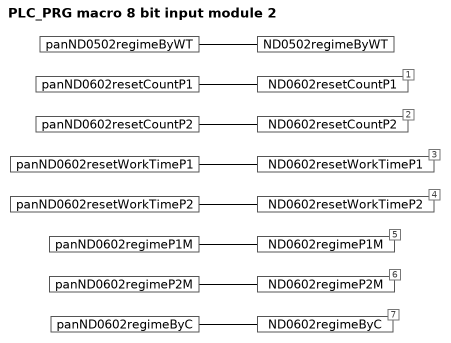
[picture p72: PLC_PRG macro 8 bit input module 2 (CFC)]
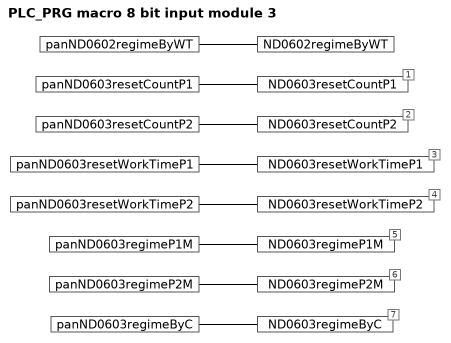
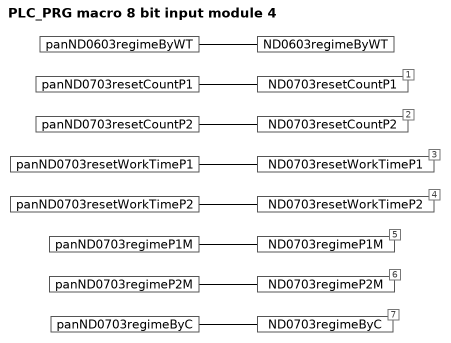
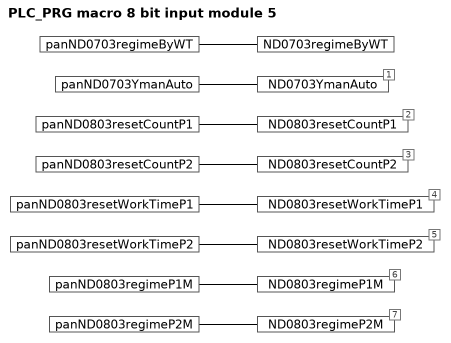
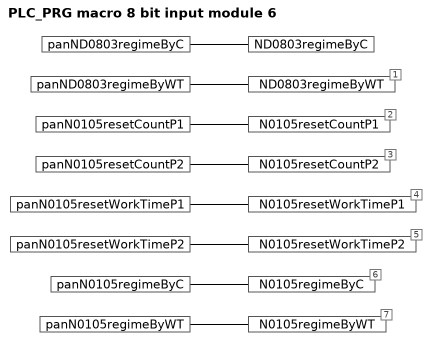
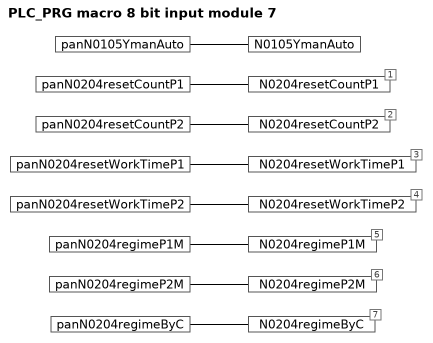
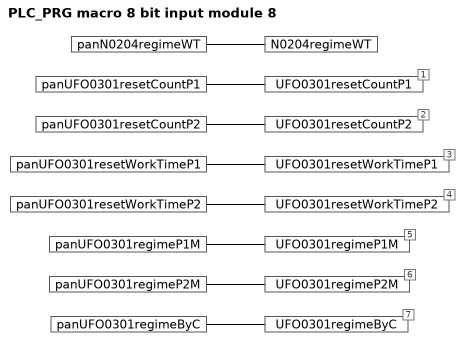
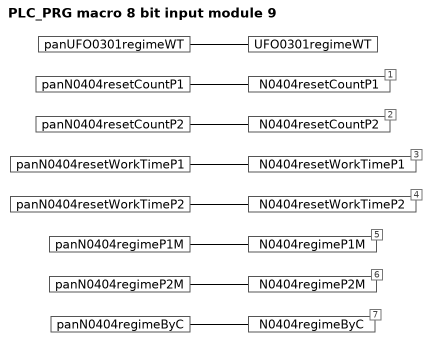
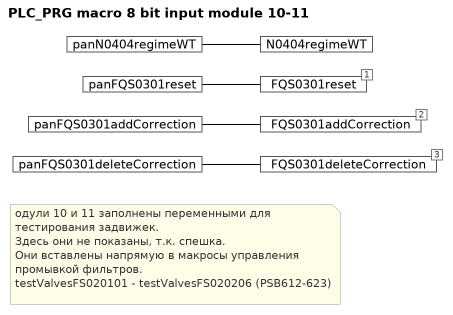
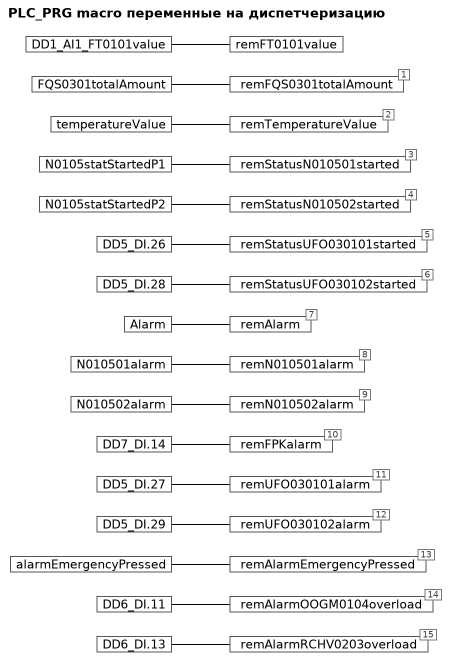
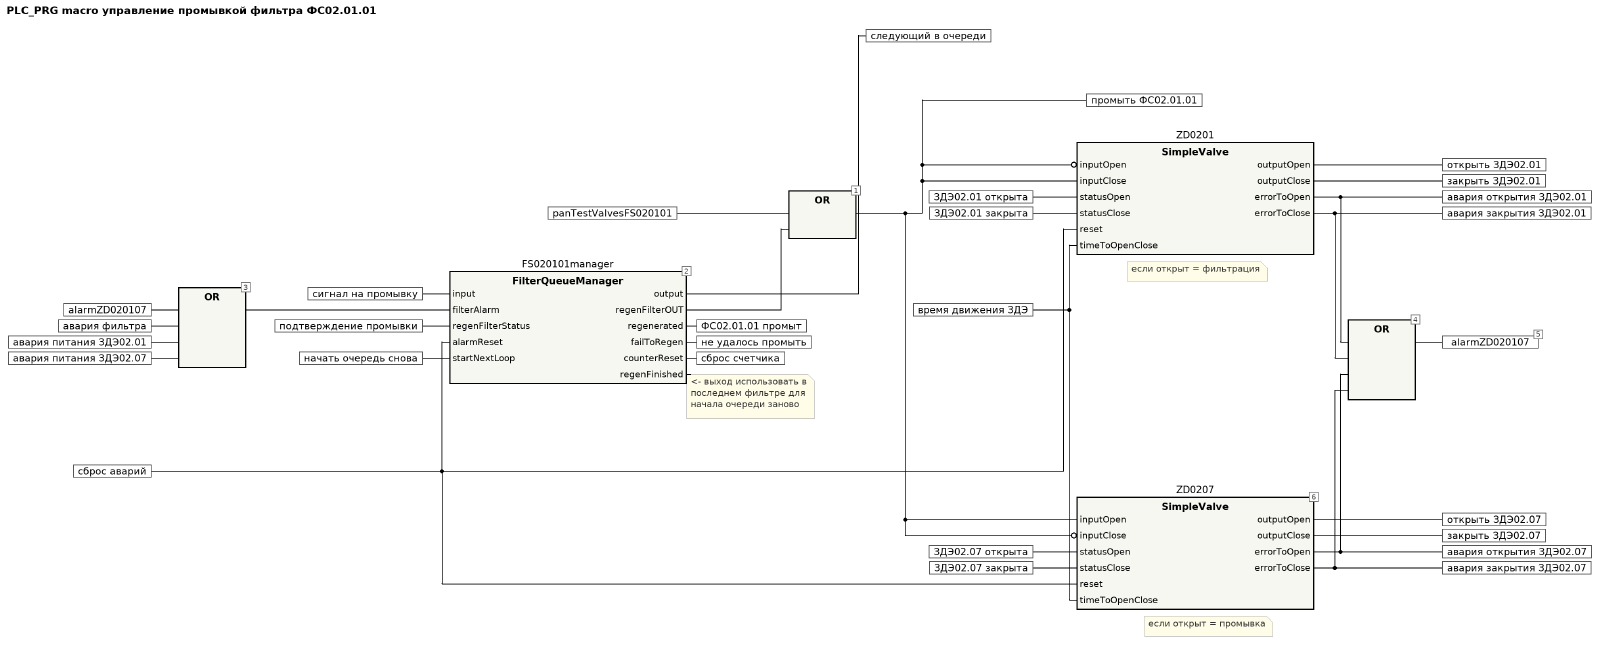
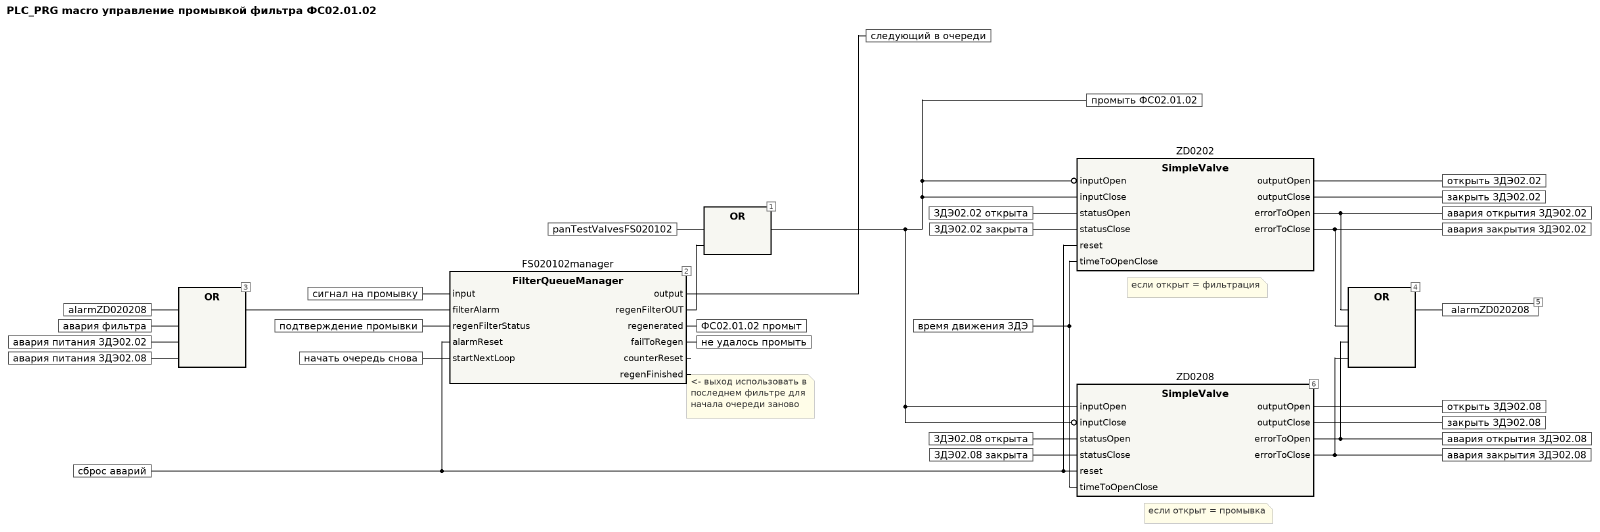
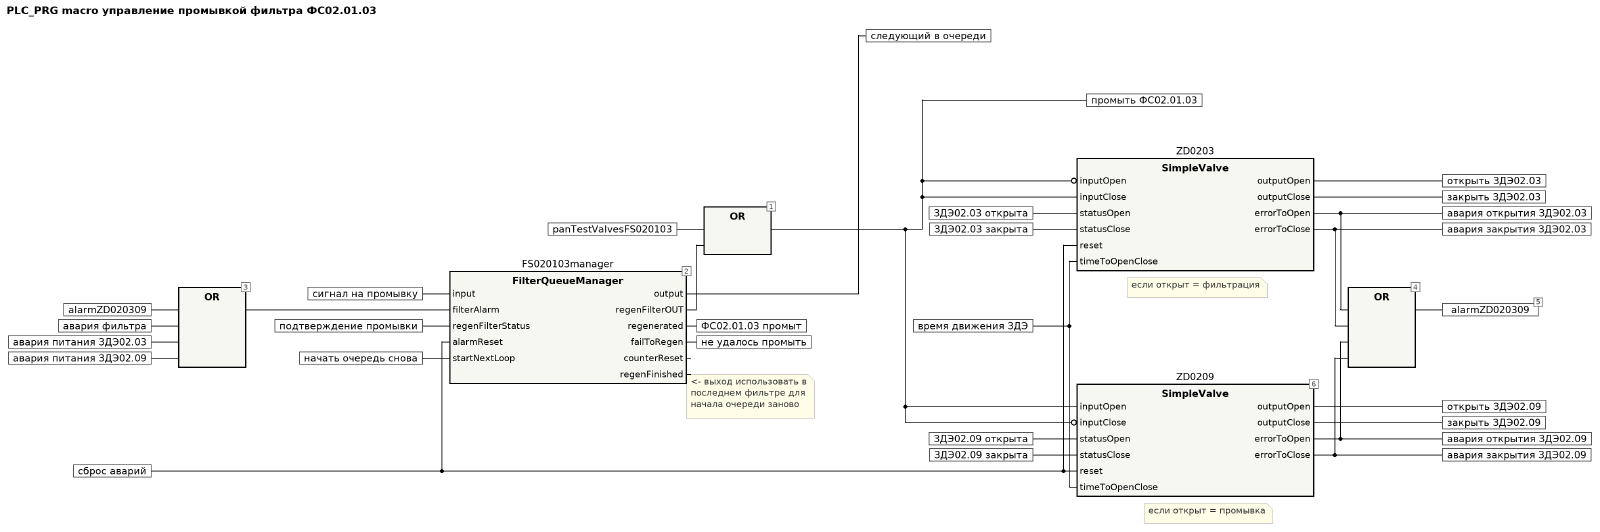
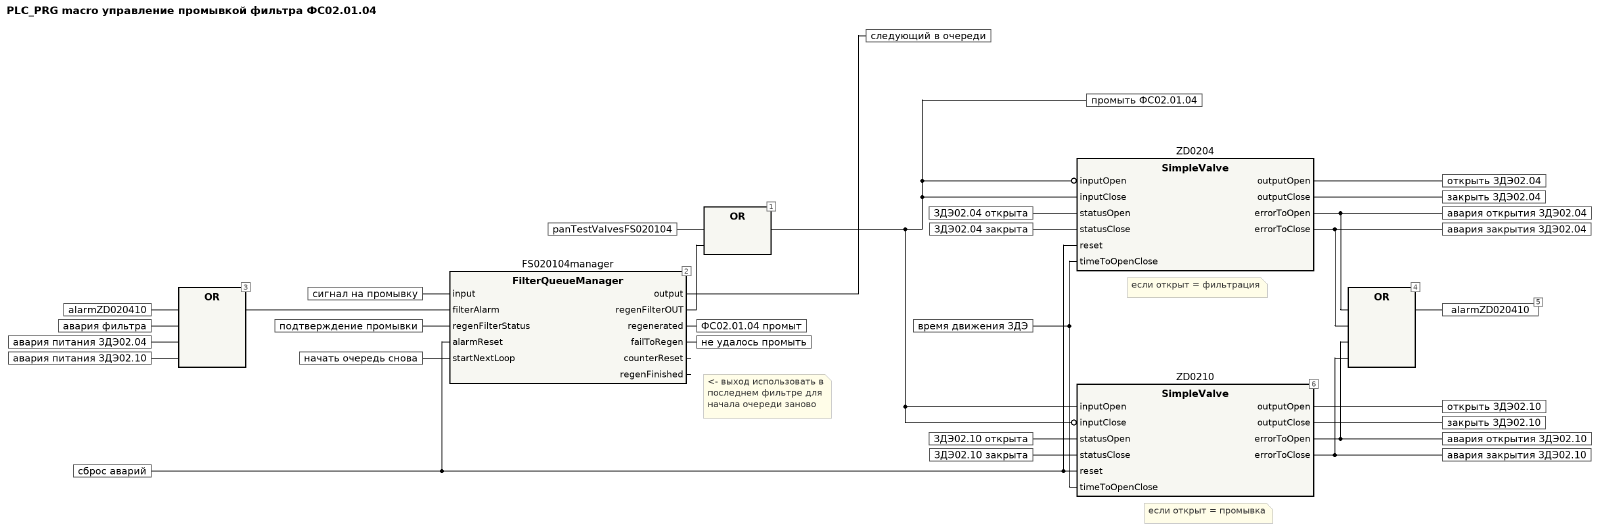
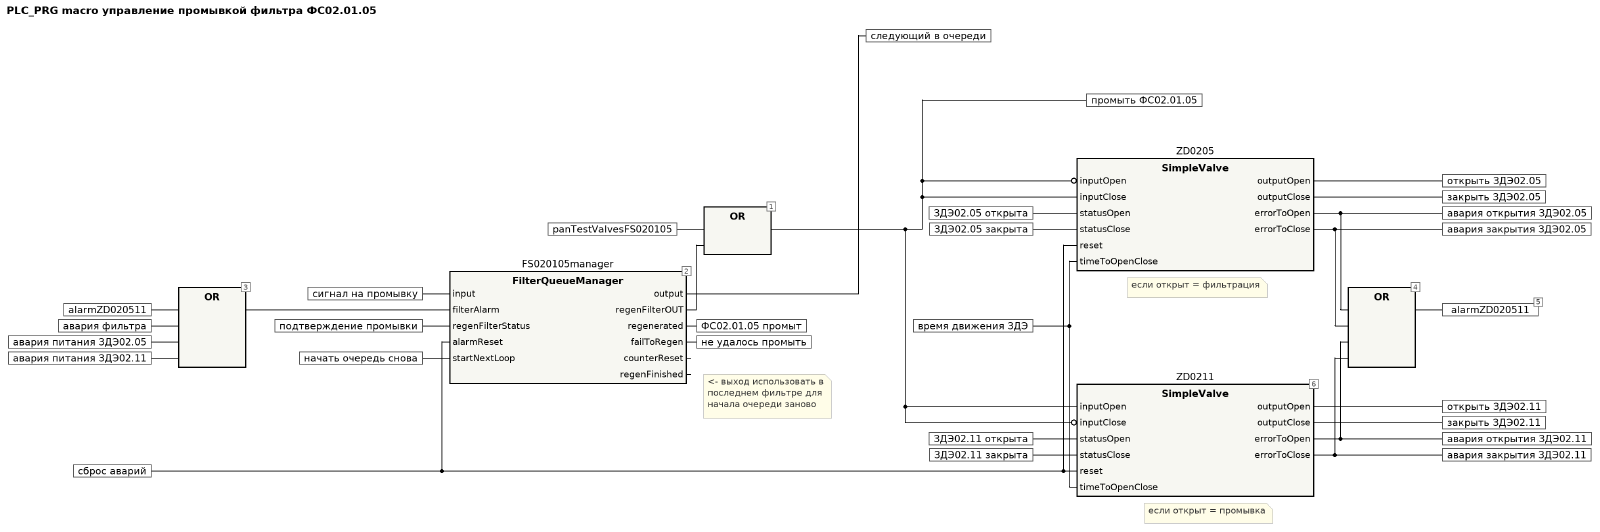
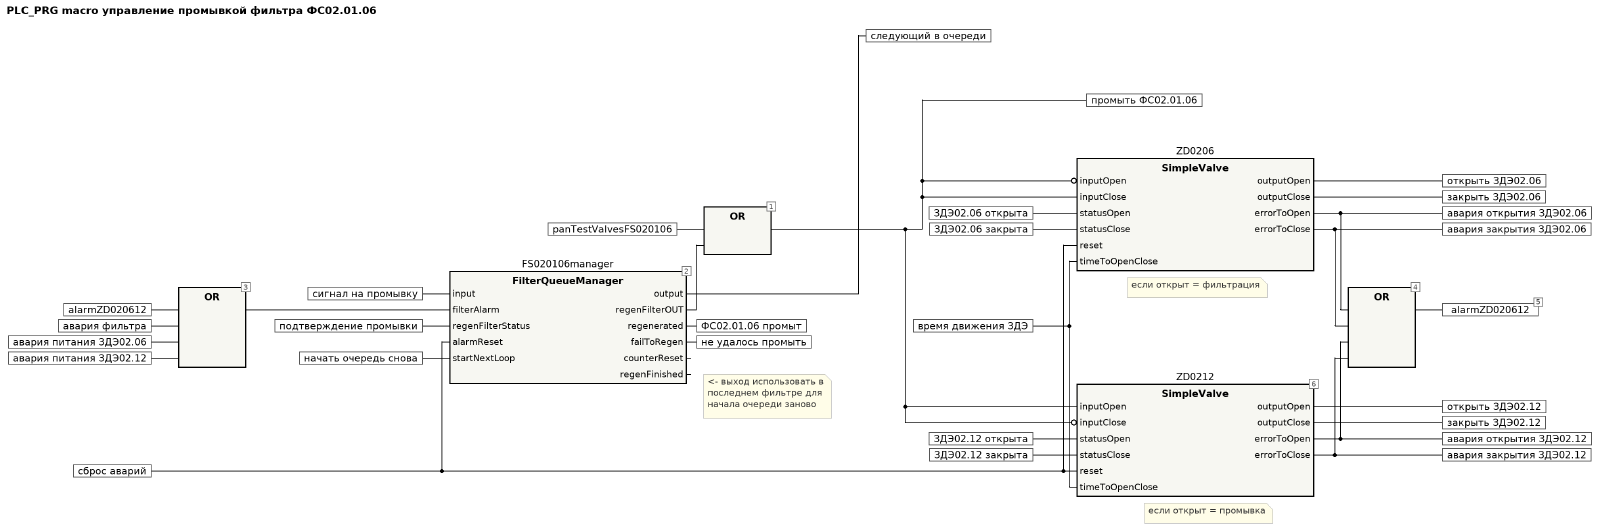
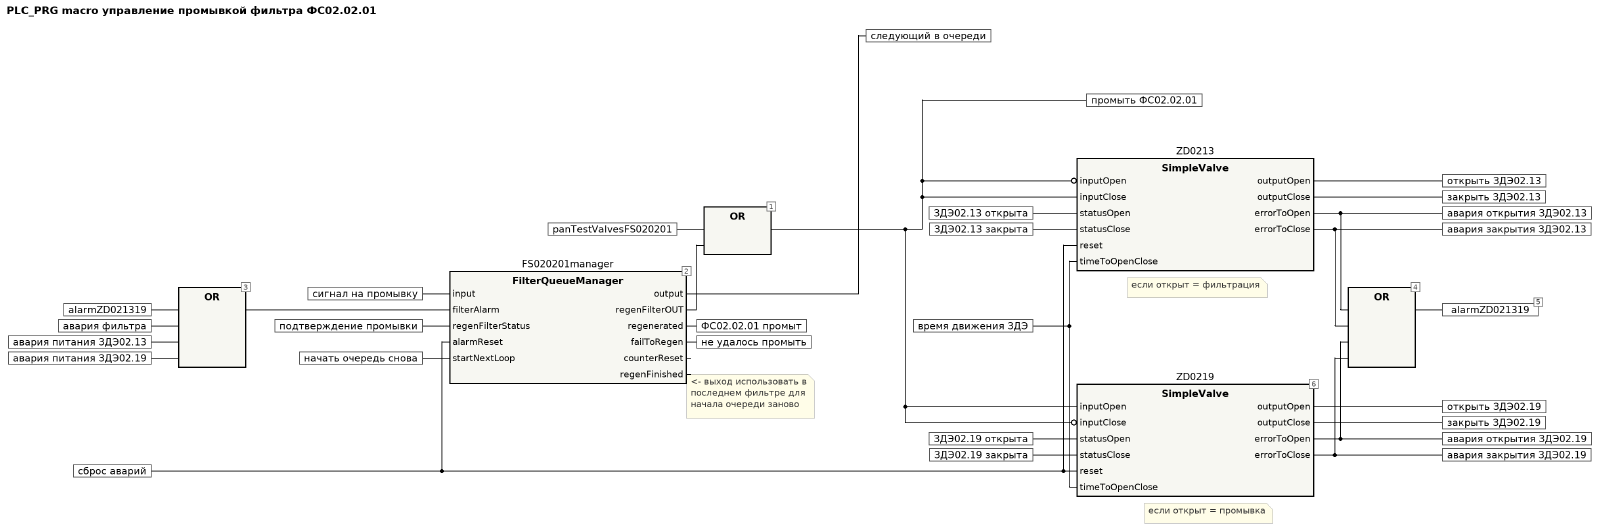
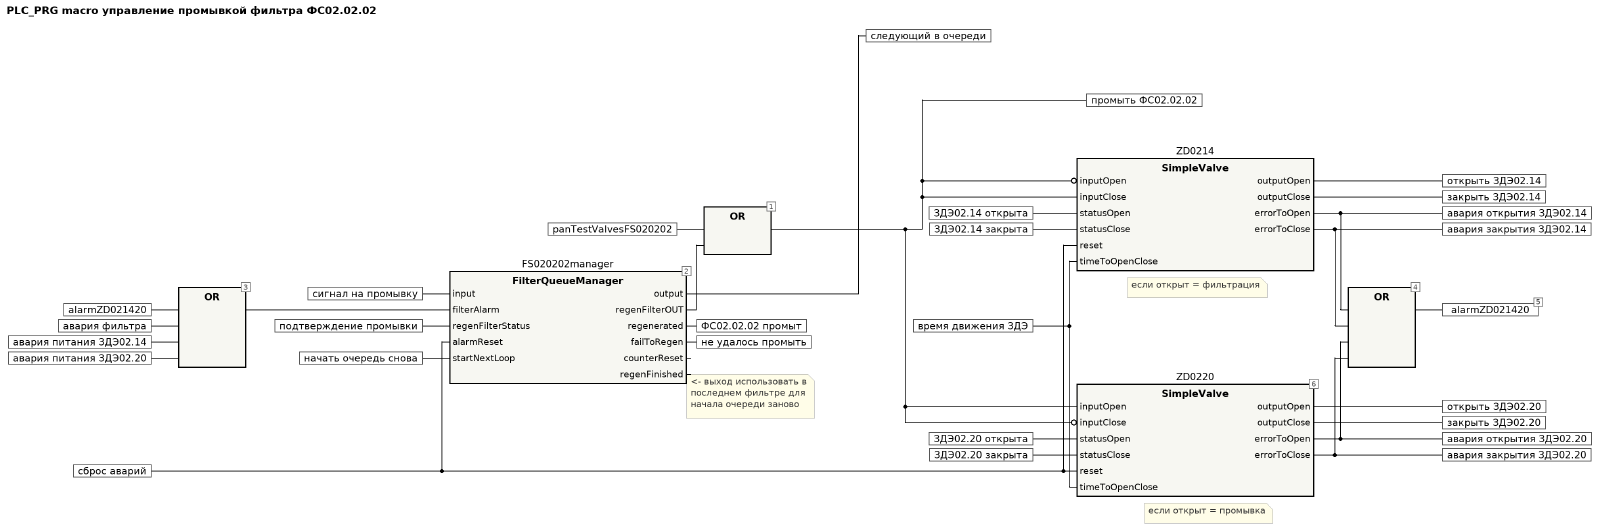
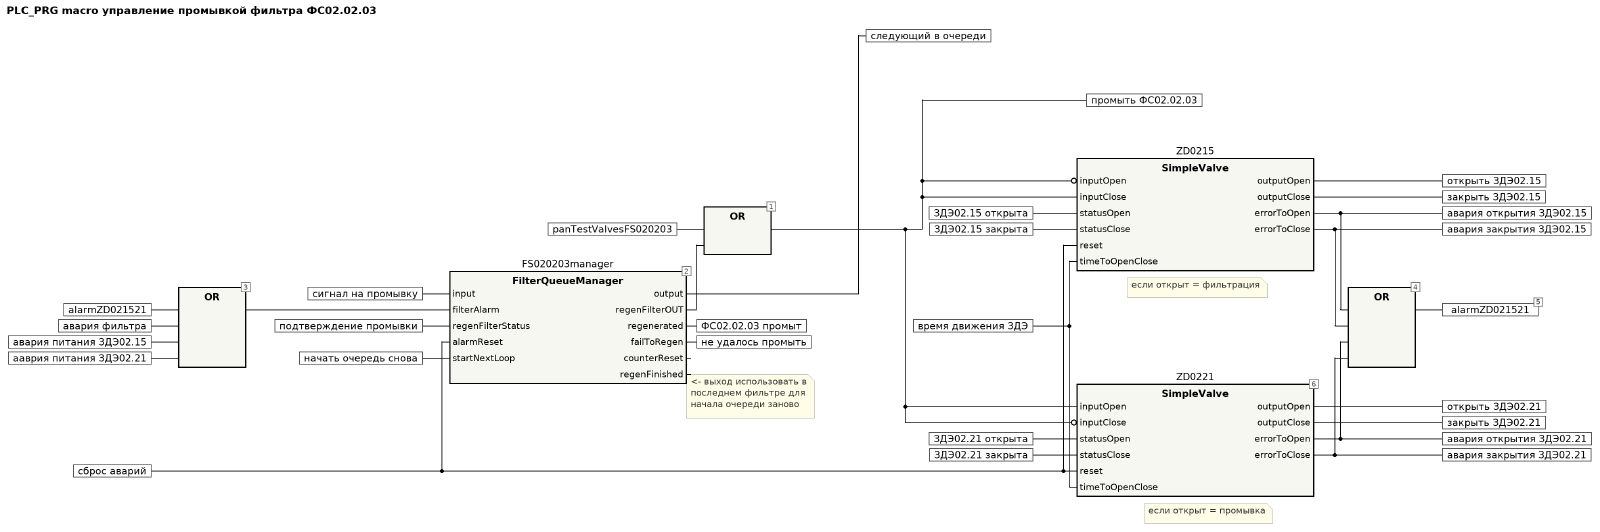
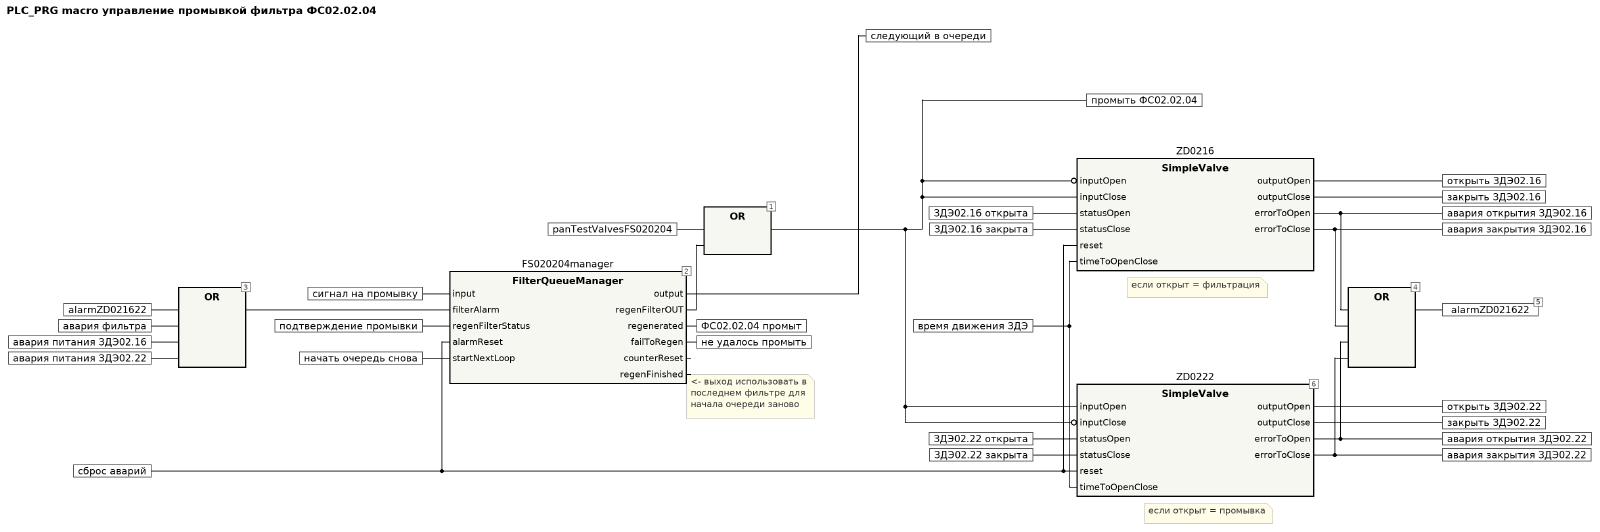
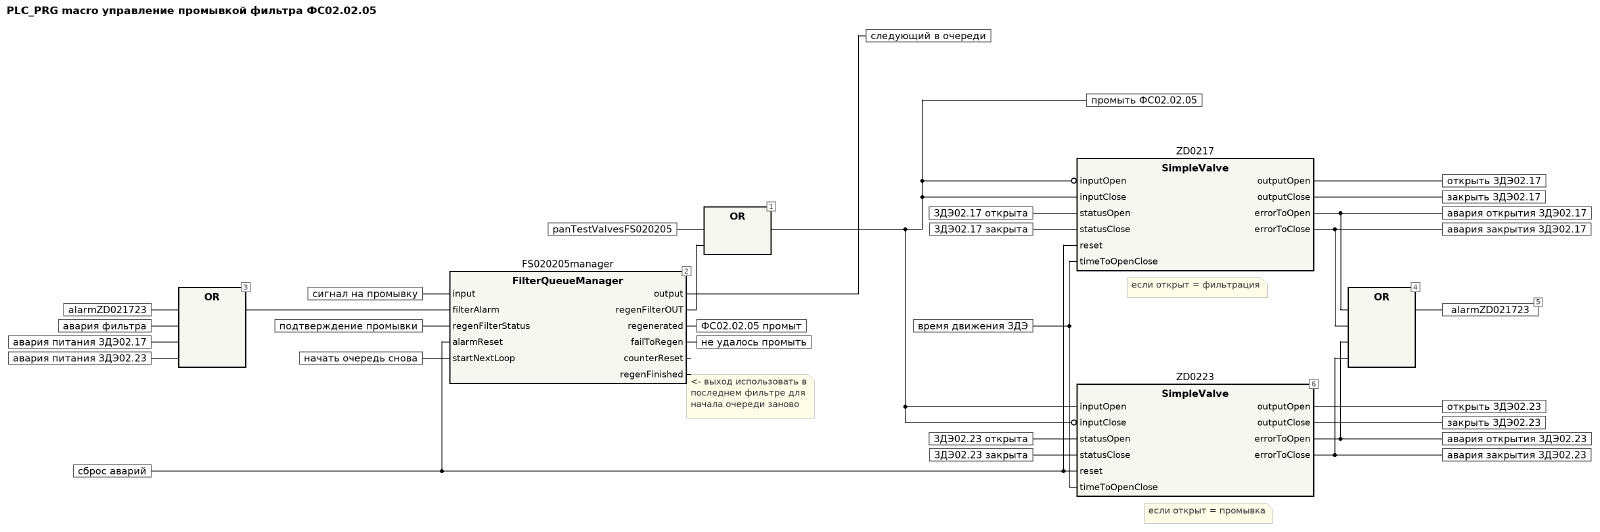
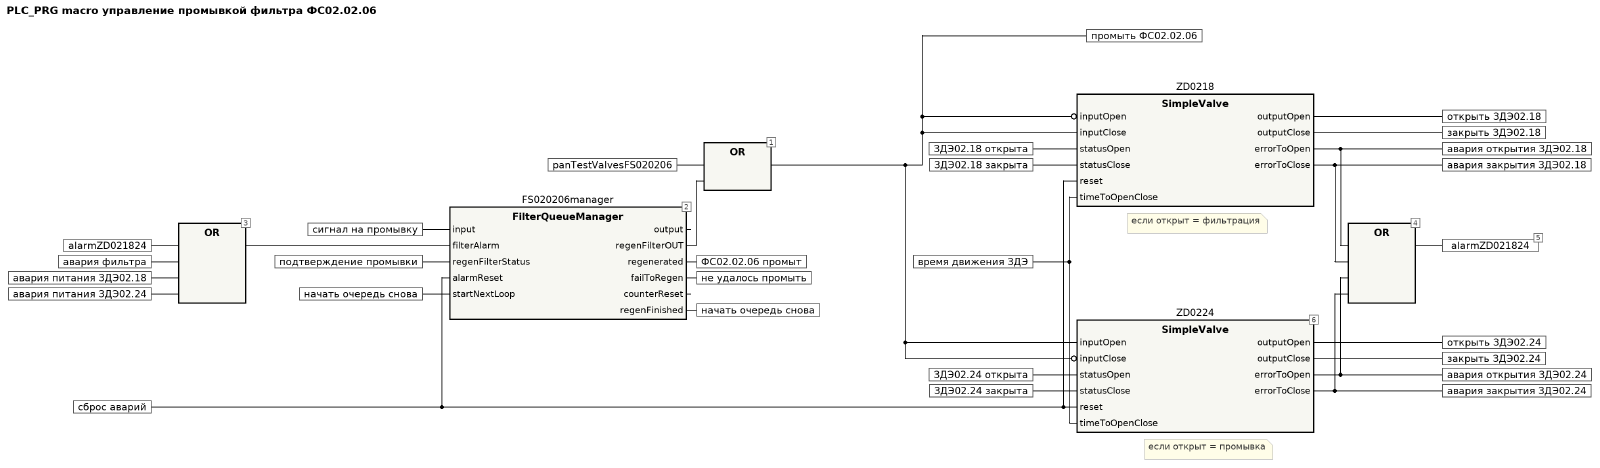
_CFC_ (* Continuous Function Chart, elements in execution order *)
(* 0 = перелив *)
(* авария обоих УФО, если проблемы / открытия/закрытия на одной из задвижек *)
(* авария питания ЗДЭ03.02 *)
(* авария питания ЗДЭ03.01 *)
(* статус-пуск Н01.05/02 *)
(* вкл КМ3 *)
(* Статус ПУСК / ЧРП Н01.05 *)
(* статус-пуск Н01.05/01 *)
(* вкл КМ2 *)
(* контроль обрыва или ошибок модулей в сети ПЛК *)
(* LSA01.02 перелив ОГМ01.04 *)
(* Нажат аварийный стоп. *)
(* авария сети (РКФ) *)
(* разрешение работы КНС / 1 = разрешено *)
(* Нажат аварийный стоп. *)
(* Блок управления разрешением работы КНС *)
(* авария сети (РКФ) *)
(* Авария питания клапанов КЭМ. *)
(* Авария питания розеток / управл.клапанов фильтров. *)
(* авария КНС *)
(* блок подачи сигнала на промывку *)
(* суммируем каждую секунду значение / мгновенного расхода в кубометрах в секунду *)
(* преобразуем расход из / кубометров в час в / кубометры в секунду *)
(* если есть расход / (больше нуля) *)
(* выдает импульс / каждую секунду *)
(* здесь мгновенный расход / в кубометрах в час (FT01.02) *)
(* Авария Н02.04/01 (0=авария) *)
(* Авария Н02.04/02 (0=авария) *)
(* промывка ФС02.01/06 *)
(* промывка ФС02.01/05 *)
(* промывка ФС02.01/04 *)
(* промывка ФС02.01/03 *)
(* промывка ФС02.01/02 *)
(* промывка ФС02.01/01 *)
(* пуск/стоп НД08.03/01 *)
(* пуск/стоп НД08.03/02 *)
(* пуск/стоп НД06.03/01 *)
(* пуск/стоп НД06.03/02 *)
(* пуск/стоп НД06.02/01 *)
(* пуск/стоп НД06.02/02 *)
(* пуск/стоп НД08.04 *)
(* пуск/стоп НД07.03/01 *)
(* пуск/стоп НД07.03/02 *)
(* авария М08.02 (УПФ) *)
(* авария М07.02 (УПЩ) *)
(* авария М06.04 (УПК) *)
(* работа М08.02 (УПФ) *)
(* работа М07.02 (УПЩ) *)
(* работа М06.04 (УПК) *)
(* Контроль, если УФО включили вручную, / а потока при этом нет. *)
(* авария УФО03.01/02 *)
(* работа УФО03.01/02 *)
(* авария УФО03.01/01 *)
(* Для подачи предостережения на пульте / оператора (при необходимости), а также / сигнализации лампой АВАРИЯ. *)
(* работа УФО03.01/01 *)
(* авария УФО03.01/02 *)
(* авария УФО03.01/01 *)
(* авария Н04.04/01 *)
(* авария Н04.04/02 *)
(* время контроля старта ФПК (по умолч.=3мин) *)
(* время работы ФПК после спада сигнала датч.осадка *)
(* запуск фильтрации *)
(* Защита от сухого хода насоса ФПК *)
(* датчик уровня осадка *)
(* Давление на входе ФПК (0...16 бар) *)
(* авария ФПК *)
(* подающий насос ФПК работает *)
(* ФПК готов к приему *)
(* ФПК не запустился *)
(* рН-метр QE01.02 на входе, / диапазон 0...14 *)
(* авария входа рН-метра QE01.01 *)
(* авария входа расходомера FT01.02 *)
(* расходомер FT01.01 на входе, / диапазон 0...600куб/час *)
(* авария НД08.04 *)
(* управление 4...20мА НД08.03/01 *)
(* пуск/стоп НД08.03/01 *)
(* пуск/стоп НД08.03/02 *)
(* управление 4...20мА НД08.03/02 *)
(* авария привода НД08.03/01 *)
(* авария привода НД08.03/02 *)
(* авария НД07.03/01 *)
(* авария НД07.03/02 *)
(* управление 4...20мА НД07.03/01 *)
(* управление 4...20мА НД07.03/02 *)
(* пуск/стоп НД07.03/01 *)
(* пуск/стоп НД07.03/02 *)
(* авария НД07.03/01 *)
(* авария НД07.03/02 *)
(* авария НД06.03/01 *)
(* авария НД06.03/02 *)
(* авария НД06.02/01 *)
(* авария НД06.02/02 *)
(* управление 4...20мА НД06.03/01 *)
(* пуск/стоп НД06.03/01 *)
(* пуск/стоп НД06.03/02 *)
(* управление 4...20мА НД06.03/02 *)
(* авария НД06.03/01 *)
(* авария НД06.03/02 *)
(* управление 4...20мА НД06.02/01 *)
(* пуск/стоп НД06.02/01 *)
(* пуск/стоп НД06.02/02 *)
(* управление 4...20мА НД06.02/02 *)
(* авария НД06.02/01 *)
(* авария НД06.02/02 *)
(* ошибка блока дозирования НД05.02 *)
(* авария входа датчика температуры *)
(* лампа АВАРИЯ *)
(* датчик температуры в помещении / (метран) диапазон: 0...+100С *)
(* управление 4...20мА НД05.02/01 *)
(* пуск/стоп НД05.02/01 *)
(* авария НД05.02/01 *)
(* авария НД05.02/02 *)
(* пуск/стоп НД05.02/02 *)
(* управление 4...20мА НД05.02/02 *)
(* АВАРИИ *)
(* авария привода НД08.03/01 *)
(* авария привода НД08.03/02 *)
(* авария НД08.04 *)
(* насос Н04.01 работает *)
(* пуск/стоп НД08.04 *)
(* управление 4...20мА НД08.04 *)
(* авария входа расходомера FT01.01 *)
(* расходомер FT01.02 на входе, / диапазон 0...600куб/час *)
(* рН-метр QE01.01 на входе, / диапазон 0...14 *)
(* авария входа рН-метра QE01.02 *)
(* сухой ход НД08.03/01 *)
(* сухой ход НД08.03/02 *)
(* сухой ход НД08.03/01 *)
(* сухой ход НД08.03/02 *)
(* LSA01.02 перелив ОГМ01.04 *)
(* Инициализирует требуемые булевые переменные / в момент старта выполнения программы. *)
(* Статус ПУСК ЧРП Н01.05 *)
(* LS01.03 - рабочий верхний уровень ОГМ01.04 автоматический пуск 01.05 *)
(* LS01.04 - нижний уровень ОГМ01.04, сухой ход Н01.05 *)
(* SA1 Ручной выбор Н01.05/01 = главный *)
(* SA1 Ручной выбор Н01.05/02 = главный *)
(* Стоп  Н01.05 (сброс самоподхвата реле) *)
(* время на создание потока *)
(* Пуск  Н01.05 *)
(* КМ1 питание ЧРП *)
(* КМ2 питание насоса 1 *)
(* КМ3 питание насоса 2 *)
(* Авария ЧРП Н01.05 *)
(* термоконтакт Н01.05/01 *)
(* термоконтакт Н01.05/02 *)
(* авария питания ЗДЭ02.25 *)
(* LSА02.01 Перелив РЧВ02.03 *)
(* Давление на входе ФПК / 0...16 бар (мах допуст.10) *)
(* Авария входа AI6 ПЛК, давл.ФПК *)
(* авария ФПК *)
(* Открыть КШЭ04.01 *)
(* статус КШЭ04.01 открыт *)
(* Закрыть КШЭ04.01 *)
(* статус КШЭ04.01 закрыт *)
(* подающий насос ФПК работает *)
(* стоп Н04.04 *)
(* пуск Н04.04/02 *)
(* пуск Н04.04/01 *)
(* авт.пуск Н04.04 *)
(* сухой ход Н04.04, 0=защита *)
(* авария Н04.04/01, 0=авария *)
(* авария Н04.04/02, 0=авария *)
(* импульсный расходомер *)
(* Авария Н02.04/01 (0=авария) *)
(* Авария Н02.04/02 (0=авария) *)
(* промывка ФС02.02/06 *)
(* промывка ФС02.02/05 *)
(* промывка ФС02.02/04 *)
(* промывка ФС02.02/03 *)
(* промывка ФС02.02/02 *)
(* промывка ФС02.02/01 *)
(* Клапан КЭМ05.01 открыт. *)
(* Клапан КЭМ06.01 открыт. *)
(* Клапан КЭМ07.01 открыт. *)
(* Клапан КЭМ08.01 открыт. *)
(* Сухой ход Н02.04 (LS02.03) 0=сух.ход *)
(* Стоп Н02.04, / сброс самоподхвата реле, / пока активно пуск - невозможен *)
(* Пуск Н02.04/01 *)
(* Пуск Н02.04/02 *)
(* текущий объем *)
(* заданный до промывки объем *)
(* 0=авария *)
(* авария (при 0) ФС02.01/06 *)
(* авария (при 0) ФС02.01/05 *)
(* авария (при 0) ФС02.01/04 *)
(* авария (при 0) ФС02.01/03 *)
(* авария (при 0) ФС02.01/02 *)
(* авария (при 0) ФС02.01/01 *)
(* авария (при 0) ФС02.02/06 *)
(* авария (при 0) ФС02.02/05 *)
(* авария (при 0) ФС02.02/04 *)
(* авария (при 0) ФС02.02/03 *)
(* авария (при 0) ФС02.02/02 *)
(* авария (при 0) ФС02.02/01 *)
(* сброс счетчика стоков до следующей промывки *)
(* подсчет общего объема стоков, прошедшего через расходомер FT01.02 *)
(* очередь передается на 2 ступень *)
(* авария питания ЗДЭ02.01 *)
(* авария питания ЗДЭ02.02 *)
(* авария питания ЗДЭ02.03 *)
(* авария питания ЗДЭ02.04 *)
(* авария питания ЗДЭ02.05 *)
(* авария питания ЗДЭ02.06 *)
(* авария питания ЗДЭ02.07 *)
(* авария питания ЗДЭ02.08 *)
(* авария питания ЗДЭ02.09 *)
(* авария питания ЗДЭ02.10 *)
(* авария питания ЗДЭ02.11 *)
(* авария питания ЗДЭ02.12 *)
(* авария питания ЗДЭ02.13 *)
(* авария питания ЗДЭ02.14 *)
(* авария питания ЗДЭ02.15 *)
(* авария питания ЗДЭ02.16 *)
(* авария питания ЗДЭ02.17 *)
(* авария питания ЗДЭ02.18 *)
(* авария питания ЗДЭ02.19 *)
(* авария питания ЗДЭ02.20 *)
(* авария питания ЗДЭ02.21 *)
(* авария питания ЗДЭ02.22 *)
(* авария питания ЗДЭ02.23 *)
(* авария питания ЗДЭ02.24 *)
(* инвертирование сигнала, чтобы все аварии / обозначались как 1 (TRUE) *)
(* авария НД05.02/01 *)
(* авария НД05.02/02 *)
(* авария питания КШЭ04.01 *)
(* 1=открыть; 0 = закрыть *)
(* в этом макросе лежит управление режимом тестирования задвижек ЗДЭ03 / Тестирование запрещает автоматический запуск УФО от ПЛК *)
(* стоп от / панели оператора *)
#0 rTrigStartInitializer:R_TRIG(CLK: TRUE)
#1 startInitializer <= #0.Q
#2 MACRO контроль температуры в помещении(pin 1 "вход датчика температуры": DD1_AI0, pin 2 "минимально допустимая температура в помещении": maxTemperature, pin 3 "максимально допустимая температура в помещении": minTemperature)
	(* задаем границы допустимой температуры в помещении / проверяем что измеренное значение в заданном диапазоне *)
	(* не смотрим конкретный тип ошибки / (работает не точно, обрыв определяет как слишком маленькое значение) / если не равно 0 - значит на входе ошибка *)
	#3 DD1_AI0_temperature:DECODE_FLOAT(VALUE: pin 1, DEF_VALUE: -)
	#4 NE(#3._ERR, 0)
	out 2 "авария датчика температуры" <= #4
	out 1 "температура в помещении" <= #3.OUT_VALUE
	#5 REAL_TO_INT(#3.OUT_VALUE)
	#6 temperatureLimits:LIMITALARM(IN: #5, HIGH: pin 3, LOW: pin 2)
	out 3 "температура выше заданного диапазона" <= #6.O
	out 4 "температура ниже заданного диапазона" <= #6.U
	#7 temperatureLimits:LIMITALARM(IN: -, HIGH: -, LOW: -)
END_MACRO
#8 temperatureValue <= #2.out 1
#9 DD1_AI0_error <= #2.out 2
#10 alarmHighTemperature <= #2.out 3
#11 alarmLowTemperature <= #2.out 4
#12 OR(testKSHE0401, DD7_DI.13)
#13 MACRO клапан шаровый перед ФПК (КШЭ04.01)(pin 1 "сигнал "подающий насос ФПК" работает": #12, pin 2 "статус КШЭ04.01 открыт": DD9_DI.2, pin 3 "статус КШЭ04.01 закрыт": DD9_DI.3, pin 4 "сброс аварий": alarmReset, pin 5 "время на открытие/закрытие": timeToOpenCloseValve)
	#14 FPKkshe0401DelayToOpen:TON(IN: #16.outputOpen, PT: T#1s)
	out 1 "выход на открытие КШЭ04.01" <= #14.Q
	#15 FPKkshe0401DelayToClose:TON(IN: #16.outputClose, PT: T#1s)
	out 2 "выход на закрытие КШЭ04.01" <= #15.Q
	#16 FPKkshe0401:SimpleValve(inputOpen: pin 1, inputClose: #17, statusOpen: pin 2, statusClose: pin 3, reset: pin 4, timeToOpenClose: pin 5)
	#17 NOT(pin 1)
	out 3 "авария на открытие КШЭ04.01" <= #16.errorToOpen
	out 4 "авария на закрытие КШЭ04.01" <= #16.errorToClose
END_MACRO
#18 DD4_DO.2 <= #13.out 1
#19 DD4_DO.3 <= #13.out 2
#20 FPKkshe0401errorToOpen <= #13.out 3
#21 FPKkshe0401errorToClose <= #13.out 4
#22 OR(DD1_AI0_error, DD1_AI1_error, DD1_AI2_error, DD1_AI3_error, DD1_AI4_error, alarmHighTemperature, alarmLowTemperature, ND0502dosingError, ND0602dosingError, ND0603dosingError, ND0803dosingError, ND0804dosingError, DD1_DI6, DD1_DI7, N010501alarm, N010502alarm, ZDE0225errorToOpen, ZDE0225errorToClose, DD7_DI.14, FPKnotStarted, DD1_AI5_error, FPKkshe0401errorToOpen, FPKkshe0401errorToClose, DD5_DI.27, DD5_DI.29, filterFailToRegen020101, errorToOpenZD0201, errorToCloseZD0201, errorToOpenZD0207, errorToCloseZD0207, filterFailToRegen020102, errorToOpenZD0202, errorToCloseZD0202, errorToOpenZD0208, errorToCloseZD0208, filterFailToRegen020103, errorToOpenZD0203, errorToCloseZD0203, errorToOpenZD0209, errorToCloseZD0209, filterFailToRegen020104, errorToOpenZD0204, errorToCloseZD0204, errorToOpenZD0210, errorToCloseZD0210, filterFailToRegen020105, errorToOpenZD0205, errorToCloseZD0205, errorToOpenZD0211, errorToCloseZD0211, filterFailToRegen020106, errorToOpenZD0206, errorToCloseZD0206, errorToOpenZD0212, errorToCloseZD0212, filterFailToRegen020201, errorToOpenZD0213, errorToCloseZD0213, errorToOpenZD0219, errorToCloseZD0219, filterFailToRegen020202, errorToOpenZD0214, errorToCloseZD0214, errorToOpenZD0220, errorToCloseZD0220, filterFailToRegen020203, errorToOpenZD0215, errorToCloseZD0215, errorToOpenZD0221, errorToCloseZD0221, filterFailToRegen020204, errorToOpenZD0216, errorToCloseZD0216, errorToOpenZD0222, errorToCloseZD0222, filterFailToRegen020205, errorToOpenZD0217, errorToCloseZD0217, errorToOpenZD0223, errorToCloseZD0223, filterFailToRegen020206, errorToOpenZD0218, errorToCloseZD0218, errorToOpenZD0224, errorToCloseZD0224, alarmPLKnetwork, alarmND050201, alarmND050202, alarmND060201, alarmND060202, alarmND060301, alarmND060302, alarmND070301, alarmND070302, alarmND080301, alarmND080302, alarmND0804, alarmOGM0104overload, alarmRCHV0203overload, alarmN040402, alarmN040401, alarmM0604, alarmM0702, alarmM0802, alarmN020401, alarmN020402, alarmFS020101, alarmFS020102, alarmFS020103, alarmFS020104, alarmFS020105, alarmFS020106, alarmFS020201, alarmFS020202, alarmFS020203, alarmFS020204, alarmFS020205, alarmFS020206, alarmZDE0201power, alarmZDE0202power, alarmZDE0203power, alarmZDE0204power, alarmZDE0205power, alarmZDE0206power, alarmZDE0207power, alarmZDE0208power, alarmZDE0209power, alarmZDE0210power, alarmZDE0211power, alarmZDE0212power, alarmZDE0213power, alarmZDE0214power, alarmZDE0215power, alarmZDE0216power, alarmZDE0217power, alarmZDE0218power, alarmZDE0219power, alarmZDE0220power, alarmZDE0221power, alarmZDE0222power, alarmZDE0223power, alarmZDE0224power, alarmZDE0225power, alarmKSHE0401power, alarmKNS, alarmPowerSocketFS, alarmKEMvalvesPower, alarmEmergencyPressed, alarmRKF, errorToOpenZDE0301, errorToCloseZDE0301, errorToOpenZDE0302, errorToCloseZDE0302, alarmZDE0301power, alarmZDE0302power)
#23 DD1_DO11 <= #22
#24 alarm <= #22
#25 MACRO контроль аналогового входа DD1_AI1(pin 1 "вход": DD1_AI1)
	(* Не смотрим конкретную ошибку, / определяем,что вход неисправен без расшифровки. *)
	#26 DD1_AI1_FT0101:DECODE_FLOAT(VALUE: pin 1, DEF_VALUE: -)
	#27 NE(#26._ERR, 0)
	out 2 "авария" <= #27
	out 1 "выход" <= #26.OUT_VALUE
END_MACRO
#28 DD1_AI1_FT0101value <= #25.out 1
#29 DD1_AI1_error <= #25.out 2
#30 MACRO контроль аналогового входа DD1_AI2(pin 1 "вход": DD1_AI2)
	(* Не смотрим конкретную ошибку, / определяем,что вход неисправен без расшифровки. *)
	#31 DD1_AI2_FT0102:DECODE_FLOAT(VALUE: pin 1, DEF_VALUE: -)
	#32 NE(#31._ERR, 0)
	out 2 "авария" <= #32
	out 1 "выход" <= #31.OUT_VALUE
END_MACRO
#33 DD1_AI2_FT0102value <= #30.out 1
#34 DD1_AI2_error <= #30.out 2
#35 MACRO управление Н01.05 (поддержание заданного расхода по FT01.02)(pin 1 "статус ПУСК ЧРП (реле)": DD5_DI.4, pin 2 "LS01.03 раб.уров.": DD6_DI.12, pin 3 "LS01.04 ниж.уров.(сух.ход)": DD5_DI.0, pin 4 "SA1ручной выб.Н01.05/01-главный": DD5_DI.5, pin 5 "SA1ручной выб.Н01.05/02-главный": DD5_DI.6, pin 6 "включить режим "по кол.вкл."": N0105regimeByC, pin 7 "включить режим "по наработке"": N0105regimeByWT, pin 8 "значение расхода от FT01.02": DD1_AI2_FT0102value, pin 9 "уставка расхода": N0105flowSetValue, pin 10 "время на создание потока": N0105minFlowTime, pin 11 "Р-коэфф.": N0105koeffP, pin 12 "I-коэфф": N0105koeffI, pin 13 "Д-коэфф": N0105koeffD, pin 14 "управление ЧРП в ручн.реж.(4...20мА)": N0105YoutManual, pin 15 "переключатель управление ЧРП РУЧН/АВТ": N0105YmanAuto, pin 16 "мин.допустимый расход": N0105minFlow, pin 17 "термоконтакт Н01.05/01": DD5_DI.2, pin 18 "термоконтакт Н01.05/02": DD5_DI.3, pin 19 "авария ЧРП Н01.05": DD5_DI.1, pin 20 "сброс аварии": alarmReset, pin 21 "сброс кол-ва вкл.Н01.05/01": N0105resetCountP1, pin 22 "сброс кол-ва вкл.Н01.05/02": N0105resetCountP2, pin 23 "сброс наработки Н01.05/01": N0105resetWorkTimeP1, pin 24 "сброс наработки Н01.05/02": N0105resetWorkTimeP2)
	(* время на создание потока *)
	(* Пуск  Н01.05 *)
	(* режимы по количеству включений,  или по наработке / активны если оба входа SA1 не активны *)
	(* управление Н01.05 - поддержание / заданного расхода по FT01.02 *)
	(* по умолчанию при старте программы *)
	(* если на входе true / то нижнее значение, / иначе то, что посередине *)
	(* Если насос создает давление меньше / указанного, то авария. *)
	#36 OR(pin 2, #37.Q)
	#37 N0105startTrig:R_TRIG(CLK: pin 1)
	#38 N0105stopTrig:F_TRIG(CLK: pin 1)
	#39 N0105startTrigg:RS(SET: #36, RESET1: #41)
	#40 N0105regime:choosePumpRegime(start: #39.Q1, pump1Main: pin 4, pump2Main: pin 5, byCounter: #45, byWorkTime: #54)
	out 2 "статус режим "Н01.05/01 - главный"" <= #40.pump1MainActive
	out 3 "статус режим "Н01.05/02 - главный"" <= #40.pump2MainActive
	out 4 "статус режим "по кол-ву вкл."" <= #40.byCounterActive
	#41 OR(#38.Q, #42)
	out 5 "статус режим "по наработке"." <= #40.byWorkTimeActive
	#42 NOT(pin 3)
	#43 NOT(#39.Q1)
	out 1 "СТОП (сброс самоподхвата реле пуска ЧРП)." <= #43
	#44 AND(#53.pump1active, #63)
	out 15 "авария Н01.05/01" <= #47.Q1
	#45 AND(NOT pin 4, NOT pin 5, #51.Q1)
	#46 OR(#44, #52, NOT pin 17)
	#47 N010501alarmTrig:RS(SET: #46, RESET1: pin 20)
	#48 N010501alarm <= #47.Q1
	#49 OR(pin 6, startInitializer)
	#50 N0105regByCinit:R_TRIG(CLK: #49)
	#51 N0105regByCtrig:RS(SET: #50.Q, RESET1: #55.Q)
	#52 AND(#53.pump1active, NOT pin 19)
	#53 N0105twoPumpOneDriveManager:TwoPumpOneDriveManager(startStopPump1: #40.startPump1, startStopPump2: #40.startPump2, alarmPump1: N010501alarm, alarmPump2: N010502alarm, alarmReset: alarmReset, counterStart: #40.startByCounter, Pump1ResetCounter: pin 21, Pump2ResetCounter: pin 22, ValueToResetCounter: -, workTimeStart: #40.startByWorkTime, workTimePump1Reset: pin 23, workTimePump2Reset: pin 24, timeKM1off: -, timeKM23DelayON: -, timeKM23offDelay: -, timeReadyToStartDelay: -)
	out 6 "кол-во включений Н01.05/01" <= #53.counterPump1
	out 7 "кол-во включений Н01.05/02" <= #53.counterPump2
	out 8 "наработка Н01.05/01" <= #53.currentWorkTimePump1
	#54 AND(NOT pin 4, NOT pin 5, #56.Q1)
	out 9 "наработка Н01.05/02" <= #53.currentWorkTimePump2
	out 10 "КМ1-питание ЧРП" <= #53.DriveKM
	#55 N0105regWTinit:R_TRIG(CLK: pin 7)
	#56 N0105regWTtrig:RS(SET: #55.Q, RESET1: #50.Q)
	out 11 "КМ2-питание Н01.05/01" <= #53.pump1KM
	out 12 "КМ3-питание Н01.05/02" <= #53.pump2KM
	out 13 "пуск ЧРП (Н01.05)" <= #53.driveStart
	out 16 "авария Н01.05/02" <= #59.Q1
	#57 AND(NOT pin 19, #53.pump2active)
	#58 OR(#57, #61, NOT pin 18)
	#59 N010502alarmTrig:RS(SET: #58, RESET1: pin 20)
	#60 N010502alarm <= #59.Q1
	#61 AND(#53.pump2active, #63)
	#62 N0105timerminFlow:TON(IN: #53.driveStart, PT: pin 10)
	#63 AND(#62.Q, #64)
	#64 LE(pin 8, pin 16)
	#65 SEL(#53.driveStart, 0, #66.Y)
	out 14 "управление ЧРП (4...20мА)" <= #65
	#66 N0105pidReg:PID(ACTUAL: pin 8, SET_POINT: pin 9, KP: pin 11, TN: pin 12, TV: pin 13, Y_MANUAL: pin 14, Y_OFFSET: -, Y_MIN: 4, Y_MAX: 20, MANUAL: pin 15, RESET: #66.OVERFLOW)
END_MACRO
#67 DD4_DO.13 <= #35.out 1
#68 N0105statRegimeP1M <= #35.out 2
#69 N0105statRegimeP2M <= #35.out 3
#70 N0105statRegimeByC <= #35.out 4
#71 N0105statRegimeByWT <= #35.out 5
#72 N0105counterP1 <= #35.out 6
#73 N0105counterP2 <= #35.out 7
#74 N0105workTimeP1 <= #35.out 8
#75 N0105workTimeP2 <= #35.out 9
#76 DD2_DO.0 <= #35.out 10
#77 DD2_DO.1 <= #35.out 11
#78 DD2_DO.2 <= #35.out 12
#79 DD1_DO0 <= #35.out 13
#80 DD1_AO0 <= #35.out 14
#81 N010501alarm <= #35.out 15
#82 N010502alarm <= #35.out 16
#83 MACRO Сигналы работы с ФП04.02 (фильтр-пресс)(pin 1 "датчик уровня осадка": DD7_DI.15, pin 2 "время работы ФПК (после выкл.датч.осадка)": FPKtimeToWork, pin 3 "защита от сухого хода": DD6_DI.10, pin 4 "ошибка входа AI (обрыв)": DD1_AI5_error, pin 5 "авария ФПК": DD7_DI.14, pin 6 "фильтр-пресс готов к приему": DD7_DI.12, pin 7 "давление на входе в ФПК": DD1_AI5_FPKpressureValue, pin 8 "мах допустимое давление": FPKmaxPressureValue, pin 9 "подающий насос ФПК работает": DD7_DI.13, pin 10 "время контроля старта ФПК": FPKnotStartedTime, pin 11 "сброс аварий": alarmReset)
	(* ФПК готов к приему осадка *)
	(* LS01.01-нижн.уровень на входе ОГМ01.04 / защита от сух. хода насоса ФПК *)
	(* LES01.01-сигнал датчика уровня осадка ОГМ01.04 / запуск процесса фильтрации *)
	(* Время работы ФПК после / спада сигнала уровня осадка / по умолч.15мин. *)
	(* Давление на входе ФПК / 0...16 бар (мах допуст.10) *)
	(* максимально допустимое давление / на входе ФПК *)
	(* Условие сброса сигнала о грязном фильтр-прессе: / 1. Пропал сигнал о готовности ФПК; / 2. Появился сигнал о готовности ФПК. / Это значит, что оператор раздвигал плиты, / чистил и снова сдвигал их. *)
	#84 FPKneedToCleanResetFtrig:F_TRIG(CLK: FPKneedToCleanReset)
	#85 FPKstartTrig:RS(SET: pin 1, RESET1: #91)
	out 1 "запуск/старт ФПК" <= #85.Q1
	#86 FPKstopTimer:TOF(IN: pin 1, PT: pin 2)
	#87 FPKstopFtrig:F_TRIG(CLK: #86.Q)
	#88 AND(#85.Q1, #89)
	#89 NOT(pin 11)
	#90 AND(#85.Q1, #92.Q, #94)
	out 2 "ФПК не стартовал" <= #90
	#91 OR(#87.Q, pin 4, pin 5, #93, #95, #98.Q1)
	#92 FPKnotStartedTimer:TON(IN: #88, PT: pin 10)
	#93 NOT(pin 3)
	#94 NOT(pin 9)
	#95 NOT(pin 6)
	#96 AND(#85.Q1, #97)
	#97 GE(pin 7, pin 8)
	#98 FPKneedToCleanTrig:RS(SET: #96, RESET1: #84.Q)
	out 3 "ФПК нужно почистить!" <= #98.Q1
	#99 S FPKneedToCleanReset <= #98.Q1
	#100 FPKneedToCleanResetRtrig:R_TRIG(CLK: pin 6)
	#101 R FPKneedToCleanReset <= #100.Q
END_MACRO
#102 DD1_DO10 <= #83.out 1
#103 FPKnotStarted <= #83.out 2
#104 FPKneedToClean <= #83.out 3
#105 MACRO контроль аналогового входа DD1_AI3(pin 1 "вход": DD1_AI3)
	(* Не смотрим конкретную ошибку, / определяем,что вход неисправен без расшифровки. *)
	#106 DD1_AI3_QE0101:DECODE_FLOAT(VALUE: pin 1, DEF_VALUE: -)
	#107 NE(#106._ERR, 0)
	out 2 "авария" <= #107
	out 1 "выход" <= #106.OUT_VALUE
END_MACRO
#108 DD1_AI3_QE0101value <= #105.out 1
#109 DD1_AI3_error <= #105.out 2
#110 MACRO контроль аналогового входа DD1_AI4(pin 1 "вход": DD1_AI4)
	(* Не смотрим конкретную ошибку, / определяем,что вход неисправен без расшифровки. *)
	#111 DD1_AI4_QE0102:DECODE_FLOAT(VALUE: pin 1, DEF_VALUE: -)
	#112 NE(#111._ERR, 0)
	out 2 "авария" <= #112
	out 1 "выход" <= #111.OUT_VALUE
END_MACRO
#113 DD1_AI4_QE0102value <= #110.out 1
#114 DD1_AI4_error <= #110.out 2
#115 MACRO контроль аналогового входа DD1_AI5(pin 1 "вход": DD1_AI5)
	(* Не смотрим конкретную ошибку, / определяем,что вход неисправен без расшифровки. *)
	#116 DD1_AI5_FPK:DECODE_FLOAT(VALUE: pin 1, DEF_VALUE: -)
	#117 NE(#116._ERR, 0)
	out 2 "авария" <= #117
	out 1 "выход" <= #116.OUT_VALUE
END_MACRO
#118 DD1_AI5_FPKpressureValue <= #115.out 1
#119 DD1_AI5_error <= #115.out 2
#120 MACRO управление НД05.02 УПГ(pin 1 "вход расходомера в куб/час": DD1_AI1_FT0101value, pin 2 "max производительность НД в мл/мин": ND0502setMaxDosVal, pin 3 "задание дозирования в мл/куб": ND0502setKoefProp, pin 4 "режим:1 насос главный": ND0502regimeP1M, pin 5 "режим: 2 насос главный": ND0502regimeP2M, pin 6 "режим: по наработке": ND0502regimeByWT, pin 7 "режим: по кол-ву включений": ND0502regimeByC, pin 8 "авария 1 насоса": DD6_DI.0, pin 9 "авария 2 насоса": DD6_DI.1, pin 10 "сброс аварий": alarmReset, pin 11 "сброс счетчика включений 1 насоса": ND0502resetCountP1, pin 12 "сброс ссчетчика включений 2 насоса": ND0502resetCountP2, pin 13 "сброс наработки 1 насоса": ND0502resetWorkTimeP1, pin 14 "сброс наработки 2 насоса": ND0502resetWorkTimeP2)
	(* сигнал 4...20мА на НД05.02/02 *)
	(* сигнал 4...20мА на НД05.02/01 *)
	(* Если на входе SEL = TRUE, / то нижнее значение, / иначе - то,что посередине. *)
	#121 SEL(#128.pump1ON, 4, #122.outputValue)
	out 6 "выход 4...20мА насоса 1" <= #121
	#122 ND0502dosing:DosingPumpProportional(flowValue: pin 1, setMinPumpDosingValue: -, setMaxPumpDosingValue: pin 2, minOutputValue: -, maxOutputValue: -, setKoeffProportionality: pin 3, minFlowToStart: -)
	out 1 "ошибка блока дозирования" <= #122.dosingError
	#123 SEL(#128.pump2ON, 4, #122.outputValue)
	#124 linTrafo050202:LIN_TRAFO(IN: #123, IN_MIN: 4, IN_MAX: 20, OUT_MIN: 0, OUT_MAX: 1000)
	#125 REAL_TO_WORD(#124.OUT)
	out 7 "выход 4...20мА насоса 2" <= #125
	#126 ND0502regime:choosePumpRegime(start: #122.startDosingPump, pump1Main: pin 4, pump2Main: pin 5, byCounter: #127, byWorkTime: pin 6)
	out 2 "статус: 1 насос главный" <= #126.pump1MainActive
	out 3 "статус: 2 насос главный" <= #126.pump2MainActive
	out 4 "статус: по кол-ву включений" <= #126.byCounterActive
	#127 OR(pin 7, startInitializer)
	out 5 "статус: по наработке" <= #126.byWorkTimeActive
	#128 ND0502manager:TwoPumpManager(startStopPump1: #126.startPump1, startStopPump2: #126.startPump2, alarmPump1: #129, alarmPump2: #130, alarmReset: pin 10, counterStart: #126.startByCounter, Pump1ResetCounter: pin 11, Pump2ResetCounter: pin 12, ValueToResetCounter: -, workTimeStart: #126.startByWorkTime, workTimePump1Reset: pin 13, workTimePump2Reset: pin 14)
	out 12 "сигнал на включение насоса 1" <= #128.pump1ON
	#129 NOT(pin 8)
	out 13 "сигнал на включение насоса 2" <= #128.pump2ON
	out 8 "счетчик включений насоса 1" <= #128.counterPump1
	#130 NOT(pin 9)
	out 9 "счетчик включений насоса 2" <= #128.counterPump2
	out 10 "счетчик наработки насоса 1" <= #128.currentWorkTimePump1
	out 11 "счетчик наработки насоса 2" <= #128.currentWorkTimePump2
END_MACRO
#131 ND0502dosingError <= #120.out 1
#132 ND0502statRegimeP1M <= #120.out 2
#133 ND0502statRegimeP2M <= #120.out 3
#134 ND0502statRegimeByC <= #120.out 4
#135 ND0502statRegimeByWT <= #120.out 5
#136 DD1_AO3 <= #120.out 6
#137 DD10_AO0 <= #120.out 7
#138 ND0502counterP1 <= #120.out 8
#139 ND0502counterP2 <= #120.out 9
#140 ND0502workTimeP1 <= #120.out 10
#141 ND0502workTimeP2 <= #120.out 11
#142 DD4_DO.4 <= #120.out 12
#143 DD4_DO.5 <= #120.out 13
#144 AND(DD2_DO.1, DD5_DI.4)
#145 N0105statStartedP1 <= #144
#146 AND(DD5_DI.4, DD2_DO.2)
#147 N0105statStartedP2 <= #146
#148 MACRO Наполнение РЧВ02.03 (заслонка ЗДЭ02.25)(pin 1 "LS02.02раб.верх.уровень РЧВ": DD6_DI.14, pin 2 "LSA02.01 Перелив РЧВ": DD6_DI.13, pin 3 "статус ЗДЭ02.25 открыт": DD9_DI.0, pin 4 "статус ЗДЭ02.25 закрыт": DD9_DI.1, pin 5 "сброс аварий": alarmReset, pin 6 "время на открытие/закрытие": timeToOpenCloseValve)
	#149 OR(testZDE0225, pin 1)
	#150 NOT(pin 1)
	#151 ZDE0225:SimpleValve(inputOpen: #149, inputClose: #152, statusOpen: pin 3, statusClose: pin 4, reset: pin 5, timeToOpenClose: pin 6)
	out 1 "выход на открытие ЗДЭ02.25" <= #151.outputOpen
	#152 OR(#150, #153)
	out 2 "выход на закрытие ЗДЭ02.25" <= #151.outputClose
	out 3 "авария на открытие ЗДЭ02.25" <= #151.errorToOpen
	#153 NOT(pin 2)
	out 4 "авария на закрытие ЗДЭ02.25" <= #151.errorToClose
END_MACRO
#154 DD4_DO.0 <= #148.out 1
#155 DD4_DO.1 <= #148.out 2
#156 ZDE0225errorToOpen <= #148.out 3
#157 ZDE0225errorToClose <= #148.out 4
#158 MACRO управление Н02.04 (подача из РЧВ)(pin 1 "промывка ФС02.01/01": DD6_DI.20, pin 2 "промывка ФС02.01/02": DD6_DI.22, pin 3 "промывка ФС02.01/03": DD6_DI.24, pin 4 "промывка ФС02.01/04": DD6_DI.26, pin 5 "промывка ФС02.01/05": DD6_DI.28, pin 6 "промывка ФС02.01/06": DD6_DI.30, pin 7 "промывка ФС02.02/01": DD7_DI.0, pin 8 "промывка ФС02.02/02": DD7_DI.2, pin 9 "промывка ФС02.02/03": DD7_DI.4, pin 10 "промывка ФС02.02/04": DD7_DI.6, pin 11 "промывка ФС02.02/05": DD7_DI.8, pin 12 "промывка ФС02.02/06": DD7_DI.10, pin 13 "открыт КЭМ05.01": DD1_DI11, pin 14 "открыт КЭМ06.01": DD1_DI10, pin 15 "открыт КЭМ07.01": DD1_DI9, pin 16 "открыт КЭМ08.01": DD1_DI8, pin 17 "сухой ход Н02.04 (0=сух.ход)": DD5_DI.11, pin 18 "выбрать режим: Н02.04/01 - главный": N0204regimeP1M, pin 19 "выбрать режим: Н02.04/02 - главный": N0204regimeP2M, pin 20 "выбрать режим: по кол-ву включений": N0204regimeByC, pin 21 "выбрать режим: по наработке": N0204regimeWT, pin 22 "авария Н02.04/01 (0=авария)": DD5_DI.7, pin 23 "авария Н02.04/02 (0=авария)": DD5_DI.8, pin 24 "сброс аварий": alarmReset, pin 25 "сброс счетчика включений Н02.04/01": N0204resetCountP1, pin 26 "сброс счетчика включений Н02.04/02": N0204resetCountP2, pin 27 "сброс счетчика наработки Н02.04/01": N0204resetWorkTimeP1, pin 28 "сброс счетчика наработки Н02.04/02": N0204resetWorkTimeP2)
	(* Проверка, что фильтры 1 / ступени в регенерации (промывке) *)
	(* Проверка, что фильтры 2 / ступени в регенерации (промывке) *)
	(* Удержание сигнала на выключение насосов для / гарантированного сброса самоподхвата реле. *)
	(* Контроль открытия хотя бы одного из клапанов КЭМ *)
	(* сброс самоподхвата реле *)
	(* Защита от сухого хода Н02.04 / (LS02.03) 0=сух.ход *)
	#159 OR(pin 1, pin 2, pin 3, pin 4, pin 5, pin 6)
	#160 OR(#159, #161, #162)
	#161 OR(pin 7, pin 8, pin 9, pin 10, pin 11, pin 12)
	#162 OR(pin 13, pin 14, pin 15, pin 16)
	#163 N020401fTrigStop:F_TRIG(CLK: #170.pump1ON)
	#164 AND(#160, pin 17)
	#165 OR(#163.Q, #168.Q)
	#166 N0204stop:TOF(IN: #165, PT: T#1s)
	out 5 "стоп Н02.04" <= #166.Q
	#167 N0204chooseRegime:choosePumpRegime(start: #164, pump1Main: pin 18, pump2Main: pin 19, byCounter: #169, byWorkTime: pin 21)
	out 1 "выбран режим Н02.04/01 = главный" <= #167.pump1MainActive
	#168 N020402fTrigStop:F_TRIG(CLK: #170.pump2ON)
	out 2 "выбран режим Н02.04/02 = главный" <= #167.pump2MainActive
	out 3 "выбран режим по кол-ву включений" <= #167.byCounterActive
	#169 OR(pin 20, startInitializer)
	out 4 "выбран режим по наработке" <= #167.byWorkTimeActive
	#170 N0204manager:TwoPumpManager(startStopPump1: #167.startPump1, startStopPump2: #167.startPump2, alarmPump1: NOT pin 22, alarmPump2: NOT pin 23, alarmReset: pin 24, counterStart: #167.startByCounter, Pump1ResetCounter: pin 25, Pump2ResetCounter: pin 26, ValueToResetCounter: -, workTimeStart: #167.startByWorkTime, workTimePump1Reset: pin 27, workTimePump2Reset: pin 28)
	out 6 "пуск Н02.04/01" <= #170.pump1ON
	out 7 "пуск Н02.04/02" <= #170.pump2ON
	out 8 "счетчик включений Н02.04/01" <= #170.counterPump1
	out 9 "счетчик включений Н02.04/02" <= #170.counterPump2
	out 10 "счетчик наработки Н02.04/01" <= #170.currentWorkTimePump1
	out 11 "счетчик наработки Н02.04/02" <= #170.currentWorkTimePump2
END_MACRO
#171 N0204statRegimeP1M <= #158.out 1
#172 N0204statRegimeP2M <= #158.out 2
#173 N0204statRegimeByC <= #158.out 3
#174 N0204statRegimeWT <= #158.out 4
#175 DD1_DO1 <= #158.out 6
#176 DD1_DO2 <= #158.out 7
#177 N0204counterP1 <= #158.out 8
#178 N0204counterP2 <= #158.out 9
#179 N0204workTimeP1 <= #158.out 10
#180 N0204workTimeP2 <= #158.out 11
#181 OR(panStopN0204, #158.out 5)
#182 DD4_DO.14 <= #181
#183 MACRO управление НД06.02 УПК(pin 1 "вход расходомера в куб/час": DD1_AI2_FT0102value, pin 2 "max производительность НД в мл/мин": ND0602setMaxDosVal, pin 3 "задание дозирования в мл/куб": ND0602setKoefProp, pin 4 "режим:1 насос главный": ND0602regimeP1M, pin 5 "режим: 2 насос главный": ND0602regimeP2M, pin 6 "режим: по наработке": ND0602regimeByWT, pin 7 "режим: по кол-ву включений": ND0602regimeByC, pin 8 "авария 1 насоса": DD6_DI.2, pin 9 "авария 2 насоса": DD6_DI.3, pin 10 "сброс аварий": alarmReset, pin 11 "сброс счетчика включений 1 насоса": ND0602resetCountP1, pin 12 "сброс ссчетчика включений 2 насоса": ND0602resetCountP2, pin 13 "сброс наработки 1 насоса": ND0602resetWorkTimeP1, pin 14 "сброс наработки 2 насоса": ND0602resetWorkTimeP2)
	(* сигнал 4...20мА на НД06.02/02 *)
	(* сигнал 4...20мА на НД06.02/01 *)
	(* Если на входе SEL = TRUE, / то нижнее значение, / иначе - то,что посередине. *)
	#184 SEL(#193.pump1ON, 4, #187.outputValue)
	#185 linTraf060201:LIN_TRAFO(IN: #184, IN_MIN: 4, IN_MAX: 20, OUT_MIN: 0, OUT_MAX: 1000)
	#186 REAL_TO_WORD(#185.OUT)
	out 6 "выход 4...20мА насоса 1" <= #186
	#187 ND0602dosing:DosingPumpProportional(flowValue: pin 1, setMinPumpDosingValue: -, setMaxPumpDosingValue: pin 2, minOutputValue: -, maxOutputValue: -, setKoeffProportionality: pin 3, minFlowToStart: -)
	out 1 "ошибка блока дозирования" <= #187.dosingError
	#188 SEL(#193.pump2ON, 4, #187.outputValue)
	#189 linTraf060202:LIN_TRAFO(IN: #188, IN_MIN: 4, IN_MAX: 20, OUT_MIN: 0, OUT_MAX: 1000)
	#190 REAL_TO_WORD(#189.OUT)
	out 7 "выход 4...20мА насоса 2" <= #190
	#191 ND0602regime:choosePumpRegime(start: #187.startDosingPump, pump1Main: pin 4, pump2Main: pin 5, byCounter: #192, byWorkTime: pin 6)
	out 2 "статус: 1 насос главный" <= #191.pump1MainActive
	out 3 "статус: 2 насос главный" <= #191.pump2MainActive
	out 4 "статус: по кол-ву включений" <= #191.byCounterActive
	#192 OR(pin 7, startInitializer)
	out 5 "статус: по наработке" <= #191.byWorkTimeActive
	#193 ND0602manager:TwoPumpManager(startStopPump1: #191.startPump1, startStopPump2: #191.startPump2, alarmPump1: #194, alarmPump2: #195, alarmReset: pin 10, counterStart: #191.startByCounter, Pump1ResetCounter: pin 11, Pump2ResetCounter: pin 12, ValueToResetCounter: -, workTimeStart: #191.startByWorkTime, workTimePump1Reset: pin 13, workTimePump2Reset: pin 14)
	out 12 "сигнал на включение насоса 1" <= #193.pump1ON
	#194 NOT(pin 8)
	out 13 "сигнал на включение насоса 2" <= #193.pump2ON
	out 8 "счетчик включений насоса 1" <= #193.counterPump1
	#195 NOT(pin 9)
	out 9 "счетчик включений насоса 2" <= #193.counterPump2
	out 10 "счетчик наработки насоса 1" <= #193.currentWorkTimePump1
	out 11 "счетчик наработки насоса 2" <= #193.currentWorkTimePump2
END_MACRO
#196 ND0602dosingError <= #183.out 1
#197 ND0602statRegimeP1M <= #183.out 2
#198 ND0602statRegimeP2M <= #183.out 3
#199 ND0602statRegimeByC <= #183.out 4
#200 ND0602statRegimeByWT <= #183.out 5
#201 DD10_AO1 <= #183.out 6
#202 DD10_AO2 <= #183.out 7
#203 ND0602counterP1 <= #183.out 8
#204 ND0602counterP2 <= #183.out 9
#205 ND0602workTimeP1 <= #183.out 10
#206 ND0602workTimeP2 <= #183.out 11
#207 DD4_DO.6 <= #183.out 12
#208 DD4_DO.7 <= #183.out 13
#209 OR(errorToOpenZDE0301, errorToCloseZDE0301, errorToOpenZDE0302, errorToCloseZDE0302)
#210 OR(DD5_DI.27, #209)
#211 OR(#209, DD5_DI.29)
#212 MACRO Работа УФО03.01(pin 1 "Работа УФО03.01/01": DD5_DI.26, pin 2 "Работа УФО03.01/02": DD5_DI.28, pin 3 "Значение расхода от FT01.02": DD1_AI2_FT0102value, pin 4 "мин.допустимый расход для насосов Н01.05": N0105minFlow, pin 5 "Задержка включения УФО на создание потока": UFO0301startDelayTime, pin 6 "выбор режим: УФО03.01/01 главное": UFO0301regimeP1M, pin 7 "выбор режим: УФО03.01/02 главное": UFO0301regimeP2M, pin 8 "выбор режим: по кол-ву включений": UFO0301regimeByC, pin 9 "выбор режим: по наработке": UFO0301regimeWT, pin 10 "авария УФО03.01/01": #210, pin 11 "авария УФО03.01/02": #211, pin 12 "сброс аварий": alarmReset, pin 13 "сброс счетчика включений УФО03.01/01": UFO0301resetCountP1, pin 14 "сброс счетчика включений УФО03.01/02": UFO0301resetCountP2, pin 15 "сброс счетчика наработки УФО03.01/01": UFO0301resetWorkTimeP1, pin 16 "сброс счетчика наработки УФО03.01/02": UFO0301resetWorkTimeP2)
	(* Контроль, если УФО включили вручную, / а потока при этом нет. *)
	(* Для подачи предостережения на пульте / оператора (при необходимости), а также / сигнализации лампой АВАРИЯ. *)
	(* Задержка старта УФО *)
	(* Включаем УФО, если расходомер показывает расход больше, / чем заданный как минимально допустимый для работы насосов Н01.05. *)
	#213 OR(pin 1, pin 2)
	#214 AND(#213, #215)
	out 1 "УФО вкл без потока" <= #214
	#215 NOT(#217.Q)
	#216 GE(pin 3, pin 4)
	#217 UFO0301startDelay:TON(IN: #216, PT: pin 5)
	#218 UFO0301regimeManager:choosePumpRegime(start: #217.Q, pump1Main: pin 6, pump2Main: pin 7, byCounter: #219, byWorkTime: pin 9)
	out 2 "активен режим - главное УФО 03.01/01" <= #218.pump1MainActive
	out 3 "активен режим - главное УФО 03.01/02" <= #218.pump2MainActive
	out 4 "активен режим - по кол-ву включений" <= #218.byCounterActive
	#219 OR(startInitializer, pin 8)
	out 5 "активен режим - по наработке" <= #218.byWorkTimeActive
	#220 UFO0301manager:TwoPumpManager(startStopPump1: #218.startPump1, startStopPump2: #218.startPump2, alarmPump1: pin 10, alarmPump2: pin 11, alarmReset: pin 12, counterStart: #218.startByCounter, Pump1ResetCounter: pin 13, Pump2ResetCounter: pin 14, ValueToResetCounter: -, workTimeStart: #218.startByWorkTime, workTimePump1Reset: pin 15, workTimePump2Reset: pin 16)
	out 6 "авт. пуск УФО03.01/01" <= #220.pump1ON
	out 7 "авт. пуск УФО03.01/02" <= #220.pump2ON
	out 8 "счетчик включений УФО03.01/01" <= #220.counterPump1
	out 9 "счетчик включений УФО03.01/02" <= #220.counterPump2
	out 10 "счетчик наработки УФО03.01/01" <= #220.currentWorkTimePump1
	out 11 "счетчик наработки УФО03.01/02" <= #220.currentWorkTimePump2
END_MACRO
#221 UFO0301noFlowAttention <= #212.out 1
#222 UFO0301statRegimeP1M <= #212.out 2
#223 UFO0301statRegimeP2M <= #212.out 3
#224 UFO0301statRegimeByC <= #212.out 4
#225 UFO0301statRegimeWT <= #212.out 5
#226 UFO0301counterP1 <= #212.out 8
#227 UFO0301counterP2 <= #212.out 9
#228 UFO0301workTimeP1 <= #212.out 10
#229 UFO0301workTimeP2 <= #212.out 11
#230 MACRO работа задвижек перед УФО и автом.пуск(pin 1 "сигнал на пуск УФО03.01/01": #212.out 6, pin 2 "сигнал на пуск УФО03.01/02": #212.out 7)
	(* авт.пускУФО03.01/02 *)
	(* авт.пускУФО03.01/01 *)
	(* 1 = тест задвижек ЗДЭ / 0 = возможность автом.пуска УФО *)
	(* 1 = открыть ЗДЭ03.01 / 0 = закрыть ЗДЭ03.01 *)
	(* 1 = открыть ЗДЭ03.02 / 0 = закрыть ЗДЭ03.02 *)
	#231 NOT(testZDE03)
	#232 NOT(testZDE03)
	#233 AND(#231, #235, DD1_DI12)
	#234 DD1_DO8 <= #233
	#235 SEL(testZDE03, pin 1, manualZDE0301)
	#236 ZDE0301:SimpleValve(inputOpen: #235, inputClose: NOT #235, statusOpen: DD1_DI12, statusClose: DD1_DI13, reset: alarmReset, timeToOpenClose: timeToOpenCloseValve)
	#237 DD4_DO.16 <= #236.outputOpen
	#238 DD4_DO.17 <= #236.outputClose
	#239 errorToOpenZDE0301 <= #236.errorToOpen
	#240 errorToCloseZDE0301 <= #236.errorToClose
	#241 AND(#232, #243, DD1_DI14)
	#242 DD1_DO9 <= #241
	#243 SEL(testZDE03, pin 2, manualZDE0302)
	#244 ZDE0302:SimpleValve(inputOpen: #243, inputClose: NOT #243, statusOpen: DD1_DI14, statusClose: DD1_DI15, reset: alarmReset, timeToOpenClose: timeToOpenCloseValve)
	#245 DD4_DO.18 <= #244.outputOpen
	#246 DD4_DO.19 <= #244.outputClose
	#247 errorToOpenZDE0302 <= #244.errorToOpen
	#248 errorToCloseZDE0302 <= #244.errorToClose
END_MACRO
#249 MACRO управление НД06.03 УПК(pin 1 "вход расходомера в куб/час": DD1_AI1_FT0101value, pin 2 "max производительность НД в мл/мин": ND0603setMaxDosVal, pin 3 "задание дозирования в мл/куб": ND0603setKoefProp, pin 4 "режим:1 насос главный": ND0603regimeP1M, pin 5 "режим: 2 насос главный": ND0603regimeP2M, pin 6 "режим: по наработке": ND0603regimeByWT, pin 7 "режим: по кол-ву включений": ND0603regimeByC, pin 8 "авария 1 насоса": DD6_DI.4, pin 9 "авария 2 насоса": DD6_DI.5, pin 10 "сброс аварий": alarmReset, pin 11 "сброс счетчика включений 1 насоса": ND0603resetCountP1, pin 12 "сброс ссчетчика включений 2 насоса": ND0603resetCountP2, pin 13 "сброс наработки 1 насоса": ND0603resetWorkTimeP1, pin 14 "сброс наработки 2 насоса": ND0603resetWorkTimeP2)
	(* сигнал 4...20мА на НД06.03/02 *)
	(* сигнал 4...20мА на НД06.03/01 *)
	(* Если на входе SEL = TRUE, / то нижнее значение, / иначе - то,что посередине. *)
	#250 SEL(#259.pump1ON, 4, #253.outputValue)
	#251 linTraf060301:LIN_TRAFO(IN: #250, IN_MIN: 4, IN_MAX: 20, OUT_MIN: 0, OUT_MAX: 1000)
	#252 REAL_TO_WORD(#251.OUT)
	out 6 "выход 4...20мА насоса 1" <= #252
	#253 ND0603dosing:DosingPumpProportional(flowValue: pin 1, setMinPumpDosingValue: -, setMaxPumpDosingValue: pin 2, minOutputValue: -, maxOutputValue: -, setKoeffProportionality: pin 3, minFlowToStart: -)
	out 1 "ошибка блока дозирования" <= #253.dosingError
	#254 SEL(#259.pump2ON, 4, #253.outputValue)
	#255 linTraf060302:LIN_TRAFO(IN: #254, IN_MIN: 4, IN_MAX: 20, OUT_MIN: 0, OUT_MAX: 1000)
	#256 REAL_TO_WORD(#255.OUT)
	out 7 "выход 4...20мА насоса 2" <= #256
	#257 ND0603regime:choosePumpRegime(start: #253.startDosingPump, pump1Main: pin 4, pump2Main: pin 5, byCounter: #258, byWorkTime: pin 6)
	out 2 "статус: 1 насос главный" <= #257.pump1MainActive
	out 3 "статус: 2 насос главный" <= #257.pump2MainActive
	out 4 "статус: по кол-ву включений" <= #257.byCounterActive
	#258 OR(pin 7, startInitializer)
	out 5 "статус: по наработке" <= #257.byWorkTimeActive
	#259 ND0603manager:TwoPumpManager(startStopPump1: #257.startPump1, startStopPump2: #257.startPump2, alarmPump1: #260, alarmPump2: #261, alarmReset: pin 10, counterStart: #257.startByCounter, Pump1ResetCounter: pin 11, Pump2ResetCounter: pin 12, ValueToResetCounter: -, workTimeStart: #257.startByWorkTime, workTimePump1Reset: pin 13, workTimePump2Reset: pin 14)
	out 12 "сигнал на включение насоса 1" <= #259.pump1ON
	#260 NOT(pin 8)
	out 13 "сигнал на включение насоса 2" <= #259.pump2ON
	out 8 "счетчик включений насоса 1" <= #259.counterPump1
	#261 NOT(pin 9)
	out 9 "счетчик включений насоса 2" <= #259.counterPump2
	out 10 "счетчик наработки насоса 1" <= #259.currentWorkTimePump1
	out 11 "счетчик наработки насоса 2" <= #259.currentWorkTimePump2
END_MACRO
#262 ND0603dosingError <= #249.out 1
#263 ND0603statRegimeP1M <= #249.out 2
#264 ND0603statRegimeP2M <= #249.out 3
#265 ND0603statRegimeByC <= #249.out 4
#266 ND0603statRegimeByWT <= #249.out 5
#267 DD10_AO3 <= #249.out 6
#268 DD10_AO4 <= #249.out 7
#269 ND0603counterP1 <= #249.out 8
#270 ND0603counterP2 <= #249.out 9
#271 ND0603workTimeP1 <= #249.out 10
#272 ND0603workTimeP2 <= #249.out 11
#273 DD4_DO.8 <= #249.out 12
#274 DD4_DO.9 <= #249.out 13
#275 MACRO управление Н04.04 (дренажные)(pin 1 "защита от сухого хода Н04.04": DD5_DI.18, pin 2 "автоматич.пускН04.04": DD5_DI.19, pin 3 "режим Н04.04/01 главный": N0404regimeP1M, pin 4 "режим Н04.04/02 главный": N0404regimeP2M, pin 5 "режим по кол-ву включений": N0404regimeByC, pin 6 "режим по наработке": N0404regimeWT, pin 7 "авария Н04.04/01": DD5_DI.15, pin 8 "авария Н04.04/02": DD5_DI.14, pin 9 "сброс аварий": alarmReset, pin 10 "сброс счетчика включений Н04.04/01": N0404resetCountP1, pin 11 "сброс счетчика включений Н04.04/02": N0404resetCountP2, pin 12 "сброс счетчика наработки Н04.04/01": N0404resetWorkTimeP1, pin 13 "сброс счетчика наработки Н04.04/02": N0404resetWorkTimeP2)
	(* сбрасывает самоподхват пускового реле *)
	(* Излишняя перестраховка по сухому ходу, / на уровне реле уже все отрабатывается. *)
	(* насосы имеют электрическую блокировку / от одновременного включения *)
	(* от поплавка *)
	(* сухой ход Н04.04 / 0=защита *)
	(* 0=авария *)
	#276 NOT(pin 1)
	out 1 "стоп Н04.04" <= #276
	#277 AND(pin 1, pin 2)
	#278 N0401choosePumpRegime:choosePumpRegime(start: #277, pump1Main: pin 3, pump2Main: pin 4, byCounter: #279, byWorkTime: pin 6)
	out 2 "выбран режим: Н04.04/01 главный" <= #278.pump1MainActive
	out 3 "выбран режим: Н04.04/02 главный" <= #278.pump2MainActive
	out 4 "выбран режим: по кол-ву включений" <= #278.byCounterActive
	#279 OR(startInitializer, pin 5)
	out 5 "выбран режим: по наработке" <= #278.byWorkTimeActive
	#280 N0404twoPumpManager:TwoPumpManager(startStopPump1: #278.startPump1, startStopPump2: #278.startPump2, alarmPump1: #281, alarmPump2: #282, alarmReset: pin 9, counterStart: #278.startByCounter, Pump1ResetCounter: pin 10, Pump2ResetCounter: pin 11, ValueToResetCounter: -, workTimeStart: #278.startByWorkTime, workTimePump1Reset: pin 12, workTimePump2Reset: pin 13)
	out 6 "пуск Н04.04/01" <= #280.pump1ON
	#281 NOT(pin 7)
	out 7 "пуск Н04.04/02" <= #280.pump2ON
	out 8 "счетчик кол-ва включений Н04.04/01" <= #280.counterPump1
	#282 NOT(pin 8)
	out 9 "счетчик кол-ва включений Н04.04/02" <= #280.counterPump2
	out 10 "счетчик времени наработки Н04.04/01" <= #280.currentWorkTimePump1
	out 11 "счетчик времени наработки Н04.04/02" <= #280.currentWorkTimePump2
END_MACRO
#283 DD4_DO.15 <= #275.out 1
#284 N0404statRegimeP1M <= #275.out 2
#285 N0404statRegimeP2M <= #275.out 3
#286 N0404statRegimeByC <= #275.out 4
#287 N0404statRegimeWT <= #275.out 5
#288 DD1_DO5 <= #275.out 6
#289 DD1_DO6 <= #275.out 7
#290 N0404counterP1 <= #275.out 8
#291 N0404counterP2 <= #275.out 9
#292 N0404workTimeP1 <= #275.out 10
#293 N0404workTimeP2 <= #275.out 11
#294 MACRO управление НД07.03 УПЩ (поддержка рН, ПИД-регулятор)(pin 1 "вход рН-метра QE01.01": DD1_AI3_QE0101value, pin 2 "уставка рН": ND0703pHsetValue, pin 3 "режим:1 насос главный": ND0703regimeP1M, pin 4 "режим: 2 насос главный": ND0703regimeP2M, pin 5 "режим: по наработке": ND0703regimeByWT, pin 6 "режим: по кол-ву включений": ND0703regimeByC, pin 7 "авария 1 насоса": DD6_DI.6, pin 8 "авария 2 насоса": DD6_DI.7, pin 9 "сброс аварий": alarmReset, pin 10 "сброс счетчика включений 1 насоса": ND0703resetCountP1, pin 11 "сброс счетчика включений 2 насоса": ND0703resetCountP2, pin 12 "сброс наработки 1 насоса": ND0703resetWorkTimeP1, pin 13 "сброс наработки 2 насоса": ND0703resetWorkTimeP2, pin 14 "ручное управл.выходом Y (4...20мА)": ND0703YoutManual, pin 15 "1=ручное/0=автомат.управл.": ND0703YmanAuto, pin 16 "вход расходомера FT01.01 (куб.м/час)": DD1_AI1_FT0101value, pin 17 "коэфф.I": ND0703koeffI, pin 18 "коэфф.D": ND0703koeffD, pin 19 "коэфф.Р": ND0703koeffP)
	(* сигнал 4...20мА на НД07.03/02 *)
	(* сигнал 4...20мА на НД07.03/01 *)
	(* Если на входе SEL = TRUE, / то нижнее значение, / иначе - то,что посередине. *)
	(* min расход в кубометрах в час / для неачала дозирования. *)
	#295 ND0703pidReg:PID(ACTUAL: pin 1, SET_POINT: pin 2, KP: pin 19, TN: pin 17, TV: pin 18, Y_MANUAL: pin 14, Y_OFFSET: 500, Y_MIN: 0, Y_MAX: 1000, MANUAL: pin 15, RESET: #295.OVERFLOW)
	#296 SEL(#303.pump1ON, 0, #295.Y)
	#297 REAL_TO_WORD(#296)
	out 5 "выход 4...20мА насоса 1" <= #297
	#298 SEL(#303.pump2ON, 0, #295.Y)
	#299 REAL_TO_WORD(#298)
	out 6 "выход 4...20мА насоса 2" <= #299
	#300 GE(pin 16, 10)
	#301 ND0703regime:choosePumpRegime(start: #300, pump1Main: pin 3, pump2Main: pin 4, byCounter: #302, byWorkTime: pin 5)
	out 1 "статус: 1 насос главный" <= #301.pump1MainActive
	out 2 "статус: 2 насос главный" <= #301.pump2MainActive
	out 3 "статус: по кол-ву включений" <= #301.byCounterActive
	out 4 "статус: по наработке" <= #301.byWorkTimeActive
	#302 OR(pin 6, startInitializer)
	#303 ND0703manager:TwoPumpManager(startStopPump1: #301.startPump1, startStopPump2: #301.startPump2, alarmPump1: #304, alarmPump2: #305, alarmReset: pin 9, counterStart: #301.startByCounter, Pump1ResetCounter: pin 10, Pump2ResetCounter: pin 11, ValueToResetCounter: -, workTimeStart: #301.startByWorkTime, workTimePump1Reset: pin 12, workTimePump2Reset: pin 13)
	out 11 "сигнал на включение насоса 1" <= #303.pump1ON
	#304 NOT(pin 7)
	out 12 "сигнал на включение насоса 2" <= #303.pump2ON
	out 7 "счетчик включений насоса 1" <= #303.counterPump1
	#305 NOT(pin 8)
	out 8 "счетчик включений насоса 2" <= #303.counterPump2
	out 9 "счетчик наработки насоса 1" <= #303.currentWorkTimePump1
	out 10 "счетчик наработки насоса 2" <= #303.currentWorkTimePump2
END_MACRO
#306 ND0703statRegimeP1M <= #294.out 1
#307 ND0703statRegimeP2M <= #294.out 2
#308 ND0703statRegimeByC <= #294.out 3
#309 ND0703statRegimeByWT <= #294.out 4
#310 DD10_AO5 <= #294.out 5
#311 DD10_AO6 <= #294.out 6
#312 ND0703counterP1 <= #294.out 7
#313 ND0703counterP2 <= #294.out 8
#314 ND0703workTimeP1 <= #294.out 9
#315 ND0703workTimeP2 <= #294.out 10
#316 DD4_DO.10 <= #294.out 11
#317 DD4_DO.11 <= #294.out 12
#318 MACRO импульсный счетчик FQS0301(pin 1 "вход от счетчика": DD6_DI.19, pin 2 "вес импульса счетчика": FQS0301impulsValue, pin 3 "сброс счетчика": FQS0301reset, pin 4 "величина коррекции счетчика": FQS0301correction, pin 5 "прибавить коррекцию": FQS0301addCorrection, pin 6 "вычесть коррекцию": FQS0301deleteCorrection)
	(* сброс показаний счетчика *)
	(* значение в REAL (в какой-то момент начинает / отображаться в экспоненциальной форме) *)
	(* Если в результате коррекции накопленная сумма станет меньше нуля, то она принудительно станет равна нулю. *)
	(* коррекция показаний счетчика. *)
	(* число, коорое будем прибавлять или / вычитать из накопленной суммы стоков. *)
	#319 FQS0301rTrig:R_TRIG(CLK: pin 1)
	#320 ADD(EN: #319.Q, FQS0301totalAmount, pin 2)
	out 1 "накопленная сумма стоков (REAL)" <= #320
	#321 FQS0301resetRtrig:R_TRIG(CLK: pin 3)
	#322 MOVE(EN: #321.Q, 0)
	#323 FQS0301totalAmount <= #322
	#324 FQS0301addCorrRtrig:R_TRIG(CLK: pin 5)
	#325 ADD(EN: #324.Q, FQS0301totalAmount, pin 4)
	#326 FQS0301totalAmount <= #325
	#327 FQS0301deleteCorrRtrig:R_TRIG(CLK: pin 6)
	#328 SUB(EN: #327.Q, FQS0301totalAmount, pin 4)
	#329 FQS0301totalAmount <= #328
	#330 LT(FQS0301totalAmount, 0)
	#331 MOVE(EN: #330, 0)
	#332 FQS0301totalAmount <= #331
END_MACRO
#333 FQS0301totalAmount <= #318.out 1
#334 MACRO управление НД08.03 УПФ(pin 1 "вход расходомера в куб/час": DD1_AI1_FT0101value, pin 2 "max производительность НД в мл/мин": ND0803setMaxDosVal, pin 3 "задание дозирования в мл/куб": ND0803setKoefProp, pin 4 "режим:1 насос главный": ND0803regimeP1M, pin 5 "режим: 2 насос главный": ND0803regimeP2M, pin 6 "режим: по наработке": ND0803regimeByWT, pin 7 "режим: по кол-ву включений": ND0803regimeByC, pin 8 "авария 1 насоса": DD5_DI.12, pin 9 "авария 2 насоса": DD5_DI.13, pin 10 "сброс аварий": alarmReset, pin 11 "сброс счетчика включений 1 насоса": ND0803resetCountP1, pin 12 "сброс ссчетчика включений 2 насоса": ND0803resetCountP2, pin 13 "сброс наработки 1 насоса": ND0803resetWorkTimeP1, pin 14 "сброс наработки 2 насоса": ND0803resetWorkTimeP2, pin 15 "сухой ход 1 насоса": DD1_DI6, pin 16 "сухой ход 2 насоса": DD1_DI7)
	(* сигнал 4...20мА на НД08.03/02 *)
	(* сигнал 4...20мА на НД08.03/01 *)
	(* Если на входе SEL = TRUE, / то нижнее значение, / иначе - то,что посередине. *)
	#335 SEL(#344.pump1ON, 0, #336.outputValue)
	out 6 "выход 4...20мА насоса 1" <= #335
	#336 ND0803dosing:DosingPumpProportional(flowValue: pin 1, setMinPumpDosingValue: -, setMaxPumpDosingValue: pin 2, minOutputValue: -, maxOutputValue: -, setKoeffProportionality: pin 3, minFlowToStart: -)
	out 1 "ошибка блока дозирования" <= #336.dosingError
	#337 SEL(#344.pump2ON, 0, #336.outputValue)
	out 7 "выход 4...20мА насоса 2" <= #337
	#338 ND0803regime:choosePumpRegime(start: #336.startDosingPump, pump1Main: pin 4, pump2Main: pin 5, byCounter: #339, byWorkTime: pin 6)
	out 2 "статус: 1 насос главный" <= #338.pump1MainActive
	out 3 "статус: 2 насос главный" <= #338.pump2MainActive
	out 4 "статус: по кол-ву включений" <= #338.byCounterActive
	#339 OR(pin 7, startInitializer)
	out 5 "статус: по наработке" <= #338.byWorkTimeActive
	out 12 "сигнал на включение насоса 1" <= #344.pump1ON
	#340 NOT(pin 8)
	#341 OR(#340, pin 15)
	out 13 "сигнал на включение насоса 2" <= #344.pump2ON
	#342 NOT(pin 9)
	#343 OR(#342, pin 16)
	#344 ND0803manager:TwoPumpManager(startStopPump1: #338.startPump1, startStopPump2: #338.startPump2, alarmPump1: #341, alarmPump2: #343, alarmReset: pin 10, counterStart: #338.startByCounter, Pump1ResetCounter: pin 11, Pump2ResetCounter: pin 12, ValueToResetCounter: -, workTimeStart: #338.startByWorkTime, workTimePump1Reset: pin 13, workTimePump2Reset: pin 14)
	out 8 "счетчик включений насоса 1" <= #344.counterPump1
	out 9 "счетчик включений насоса 2" <= #344.counterPump2
	out 10 "счетчик наработки насоса 1" <= #344.currentWorkTimePump1
	out 11 "счетчик наработки насоса 2" <= #344.currentWorkTimePump2
END_MACRO
#345 ND0803dosingError <= #334.out 1
#346 ND0803statRegimeP1M <= #334.out 2
#347 ND0803statRegimeP2M <= #334.out 3
#348 ND0803statRegimeByC <= #334.out 4
#349 ND0803statRegimeByWT <= #334.out 5
#350 DD1_AO1 <= #334.out 6
#351 DD1_AO2 <= #334.out 7
#352 ND0803counterP1 <= #334.out 8
#353 ND0803counterP2 <= #334.out 9
#354 ND0803workTimeP1 <= #334.out 10
#355 ND0803workTimeP2 <= #334.out 11
#356 DD1_DO3 <= #334.out 12
#357 DD1_DO4 <= #334.out 13
#358 AND(DD1_DI5, DD1_DI4, DD6_DI.11)
#359 DD1_DO8 <= #358
#360 EQ(lastError, 0)
#361 alarmPLKnetworkDelay:TOF(IN: #360, PT: T#20s)
#362 NOT(#361.Q)
#363 alarmPLKnetwork <= #362
#364 MACRO управление НД08.04 УПФ(pin 1 "насос Н04.01 работает": DD7_DI.13, pin 2 "авария НД08.04": DD6_DI.16, pin 3 "уставкаНД08.04(0...100%)": ND0804doseValue)
	(* Преобразует сигнал 0...100 / пропорционально в 4...20мА, / в модуль АО подаем 0...1000. *)
	#365 AND(pin 1, pin 2)
	out 1 "пуск/стоп НД08.04" <= #365
	#366 ND0804linearTransformator:LIN_TRAFO(IN: pin 3, IN_MIN: 0, IN_MAX: 100, OUT_MIN: 0, OUT_MAX: 1000)
	#367 REAL_TO_WORD(#366.OUT)
	out 2 "управление НД08.04 (4...20мА)" <= #367
	out 3 "ошибка блока дозирования" <= #366.ERROR
END_MACRO
#368 DD4_DO.12 <= #364.out 1
#369 DD10_AO7 <= #364.out 2
#370 ND0804dosingError <= #364.out 3
#371 NOT(DD6_DI.0)
#372 alarmND050201 <= #371
#373 NOT(DD6_DI.23)
#374 alarmFS020102 <= #373
#375 NOT(DD9_DI.14)
#376 alarmZDE0211power <= #375
#377 NOT(DD6_DI.1)
#378 alarmND050202 <= #377
#379 NOT(DD6_DI.25)
#380 alarmFS020103 <= #379
#381 NOT(DD9_DI.15)
#382 alarmZDE0212power <= #381
#383 NOT(DD6_DI.2)
#384 alarmND060201 <= #383
#385 NOT(DD6_DI.27)
#386 alarmFS020104 <= #385
#387 NOT(DD9_DI.16)
#388 alarmZDE0213power <= #387
#389 NOT(DD6_DI.3)
#390 alarmND060202 <= #389
#391 NOT(DD6_DI.29)
#392 alarmFS020105 <= #391
#393 NOT(DD9_DI.17)
#394 alarmZDE0214power <= #393
#395 MACRO контроль включения мешалок(pin 1 "работа НД06.02/01": DD4_DO.6, pin 2 "работа НД06.02/02": DD4_DO.7, pin 3 "работа НД06.03/01": DD4_DO.8, pin 4 "работа НД06.03/02": DD4_DO.9, pin 5 "работа мешалки М06.04": DD5_DI.21, pin 6 "работа НД07.03/01": DD4_DO.10, pin 7 "работа НД07.03/02": DD4_DO.11, pin 8 "работа мешалки М07.02": DD5_DI.23, pin 9 "работа НД08.03/01": DD1_DO3, pin 10 "работа НД08.03/02": DD1_DO4, pin 11 "работа НД08.04": DD4_DO.12, pin 12 "работа мешалки М08.02": DD5_DI.25)
	#396 OR(pin 1, pin 2, pin 3, pin 4)
	#397 AND(#396, #398)
	out 1 "дозирования при выключенной М06.04" <= #397
	#398 NOT(pin 5)
	#399 OR(pin 6, pin 7)
	#400 AND(#399, #401)
	out 2 "дозирования при выключенной М07.02" <= #400
	#401 NOT(pin 8)
	#402 OR(pin 9, pin 10, pin 11)
	#403 AND(#402, #404)
	out 3 "дозирования при выключенной М08.02" <= #403
	#404 NOT(pin 12)
END_MACRO
#405 M0604attention <= #395.out 1
#406 M0702attention <= #395.out 2
#407 M0802attention <= #395.out 3
#408 NOT(DD6_DI.4)
#409 alarmND060301 <= #408
#410 NOT(DD6_DI.31)
#411 alarmFS020106 <= #410
#412 NOT(DD9_DI.18)
#413 alarmZDE0215power <= #412
#414 NOT(DD6_DI.5)
#415 alarmND060302 <= #414
#416 NOT(DD7_DI.1)
#417 alarmFS020201 <= #416
#418 NOT(DD9_DI.19)
#419 alarmZDE0216power <= #418
#420 NOT(DD6_DI.6)
#421 alarmND070301 <= #420
#422 NOT(DD7_DI.3)
#423 alarmFS020202 <= #422
#424 NOT(DD9_DI.20)
#425 alarmZDE0217power <= #424
#426 NOT(DD6_DI.7)
#427 alarmND070302 <= #426
#428 NOT(DD7_DI.5)
#429 alarmFS020203 <= #428
#430 NOT(DD9_DI.21)
#431 alarmZDE0218power <= #430
#432 NOT(DD5_DI.12)
#433 alarmND080301 <= #432
#434 NOT(DD7_DI.7)
#435 alarmFS020204 <= #434
#436 NOT(DD9_DI.22)
#437 alarmZDE0219power <= #436
#438 NOT(DD5_DI.13)
#439 alarmND080302 <= #438
#440 NOT(DD7_DI.9)
#441 alarmFS020205 <= #440
#442 NOT(DD9_DI.23)
#443 alarmZDE0220power <= #442
#444 NOT(DD6_DI.16)
#445 alarmND0804 <= #444
#446 NOT(DD7_DI.11)
#447 alarmFS020206 <= #446
#448 NOT(DD9_DI.24)
#449 alarmZDE0221power <= #448
#450 NOT(DD6_DI.11)
#451 alarmOGM0104overload <= #450
#452 NOT(DD9_DI.4)
#453 alarmZDE0201power <= #452
#454 NOT(DD9_DI.25)
#455 alarmZDE0222power <= #454
#456 MACRO переменные для обмена с панелью()
	#457 MACRO PSW регистры на передачу в панель (отображение)()
		(* PSW регистры на передачу в панель (отображение) *)
		(* panFQS0301totalAmount - переменная отображена сразу на выходе соответствующего макроса (учет очищенных стоков). / Здесь не хранится. *)
		#458 panFT0101value <= DD1_AI1_FT0101value
		#459 panQE0101value <= DD1_AI3_QE0101value
		#460 panFT0102value <= DD1_AI2_FT0102value
		#461 panQE0102value <= DD1_AI4_QE0102value
		#462 panFPKpressureValue <= DD1_AI5_FPKpressureValue
		#463 panFQS0301total <= FQS0301totalAmount
		#464 panTemperature <= temperatureValue
		#465 MACRO Время наработки и кол-во включений агрегатов()
			#466 workTimeND050201:TimeFromWorkTime(input: ND0502workTimeP1)
			#467 panND050201workDays <= #466.days
			#468 panND050201workHours <= #466.hours
			#469 panND050201workMinutes <= #466.minutes
			#470 panND050201workSeconds <= #466.seconds
			#471 workTimeND050202:TimeFromWorkTime(input: ND0502workTimeP2)
			#472 panND050202workDays <= #471.days
			#473 panND050202workHours <= #471.hours
			#474 panND050202workMinutes <= #471.minutes
			#475 panND050202workSeconds <= #471.seconds
			#476 panND0502counterP1 <= ND0502counterP1
			#477 panND0502counterP2 <= ND0502counterP2
			#478 workTimeND060201:TimeFromWorkTime(input: ND0602workTimeP1)
			#479 panND060201workDays <= #478.days
			#480 panND060201workHours <= #478.hours
			#481 panND060201workMinutes <= #478.minutes
			#482 panND060201workSeconds <= #478.seconds
			#483 workTimeND060202:TimeFromWorkTime(input: ND0602workTimeP2)
			#484 panND060202workDays <= #483.days
			#485 panND060202workHours <= #483.hours
			#486 panND060202workMinutes <= #483.minutes
			#487 panND060202workSeconds <= #483.seconds
			#488 panND0602counterP1 <= ND0602counterP1
			#489 panND0602counterP2 <= ND0602counterP2
			#490 workTimeND060301:TimeFromWorkTime(input: ND0603workTimeP1)
			#491 panND060301workDays <= #490.days
			#492 panND060301workHours <= #490.hours
			#493 panND060301workMinutes <= #490.minutes
			#494 panND060301workSeconds <= #490.seconds
			#495 workTimeND060302:TimeFromWorkTime(input: ND0603workTimeP2)
			#496 panND060302workDays <= #495.days
			#497 panND060302workHours <= #495.hours
			#498 panND060302workMinutes <= #495.minutes
			#499 panND060302workSeconds <= #495.seconds
			#500 panND0603counterP1 <= ND0603counterP1
			#501 panND0603counterP2 <= ND0603counterP2
			#502 workTimeND070301:TimeFromWorkTime(input: ND0703workTimeP1)
			#503 panND070301workDays <= #502.days
			#504 panND070301workHours <= #502.hours
			#505 panND070301workMinutes <= #502.minutes
			#506 panND070301workSeconds <= #502.seconds
			#507 workTimeND070302:TimeFromWorkTime(input: ND0703workTimeP2)
			#508 panND070302workDays <= #507.days
			#509 panND070302workHours <= #507.hours
			#510 panND070302workMinutes <= #507.minutes
			#511 panND070302workSeconds <= #507.seconds
			#512 panND0703counterP1 <= ND0703counterP1
			#513 panND0703counterP2 <= ND0703counterP2
			#514 workTimeND080301:TimeFromWorkTime(input: ND0803workTimeP1)
			#515 panND080301workDays <= #514.days
			#516 panND080301workHours <= #514.hours
			#517 panND080301workMinutes <= #514.minutes
			#518 panND080301workSeconds <= #514.seconds
			#519 workTimeND080302:TimeFromWorkTime(input: ND0803workTimeP2)
			#520 panND080302workDays <= #519.days
			#521 panND080302workHours <= #519.hours
			#522 panND080302workMinutes <= #519.minutes
			#523 panND080302workSeconds <= #519.seconds
			#524 panND0803counterP1 <= ND0803counterP1
			#525 panND0803counterP2 <= ND0803counterP2
			#526 workTimeN010501:TimeFromWorkTime(input: N0105workTimeP1)
			#527 panN010501workDays <= #526.days
			#528 panN010501workHours <= #526.hours
			#529 panN010501workMinutes <= #526.minutes
			#530 panN010501workSeconds <= #526.seconds
			#531 workTimeN010502:TimeFromWorkTime(input: N0105workTimeP2)
			#532 panN010502workDays <= #531.days
			#533 panN010502workHours <= #531.hours
			#534 panN010502workMinutes <= #531.minutes
			#535 panN010502workSeconds <= #531.seconds
			#536 panN0105counterP1 <= N0105counterP1
			#537 panN0105counterP2 <= N0105counterP2
			#538 workTimeN020401:TimeFromWorkTime(input: N0204workTimeP1)
			#539 panN020401workDays <= #538.days
			#540 panN020401workHours <= #538.hours
			#541 panN020401workMinutes <= #538.minutes
			#542 panN020401workSeconds <= #538.seconds
			#543 workTimeN020402:TimeFromWorkTime(input: N0204workTimeP2)
			#544 panN020402workDays <= #543.days
			#545 panN020402workHours <= #543.hours
			#546 panN020402workMinutes <= #543.minutes
			#547 panN020402workSeconds <= #543.seconds
			#548 panN0204counterP1 <= N0204counterP1
			#549 panN0204counterP2 <= N0204counterP2
			#550 workTimeN040401:TimeFromWorkTime(input: N0404workTimeP1)
			#551 panN040401workDays <= #550.days
			#552 panN040401workHours <= #550.hours
			#553 panN040401workMinutes <= #550.minutes
			#554 panN040401workSeconds <= #550.seconds
			#555 workTimeN040402:TimeFromWorkTime(input: N0404workTimeP2)
			#556 panN040402workDays <= #555.days
			#557 panN040402workHours <= #555.hours
			#558 panN040402workMinutes <= #555.minutes
			#559 panN040402workSeconds <= #555.seconds
			#560 panN0404counterP1 <= N0404counterP1
			#561 panN0404counterP2 <= N0404counterP2
			#562 workTimeUFO030101:TimeFromWorkTime(input: UFO0301workTimeP1)
			#563 panUFO030101workDays <= #562.days
			#564 panUFO030101workHours <= #562.hours
			#565 panUFO030101workMinutes <= #562.minutes
			#566 panUFO030101workSeconds <= #562.seconds
			#567 workTimeUFO030102:TimeFromWorkTime(input: UFO0301workTimeP2)
			#568 panUFO030102workDays <= #567.days
			#569 panUFO030102workHours <= #567.hours
			#570 panUFO030102workMinutes <= #567.minutes
			#571 panUFO030102workSeconds <= #567.seconds
			#572 panUFO0301counterP1 <= UFO0301counterP1
			#573 panUFO0301counterP2 <= UFO0301counterP2
		END_MACRO
	END_MACRO
	#574 MACRO PSB регистры на передачу в панель (отображение)()
		(* PSB регистры на передачу в панель (отображение) *)
		#575 MACRO 8 bit output module 1()
			#576 panStartND050201 <= DD4_DO.4
			#577 panStartND050202 <= DD4_DO.5
			#578 panStartND060201 <= DD4_DO.6
			#579 panStartND060202 <= DD4_DO.7
			#580 panStartND060301 <= DD4_DO.8
			#581 panStartND060302 <= DD4_DO.9
			#582 panStartM0604 <= DD5_DI.21
			#583 panStartND070301 <= DD4_DO.10
		END_MACRO
		#584 MACRO 8 bit output module 2()
			#585 panStartND070302 <= DD4_DO.11
			#586 panStartM0702 <= DD5_DI.23
			#587 panStartND080301 <= DD1_DO3
			#588 panStartND080302 <= DD1_DO4
			#589 panStartND0804 <= DD4_DO.12
			#590 panStartM0802 <= DD5_DI.25
			#591 panStartN020401 <= DD5_DI.9
			#592 panStartN020402 <= DD5_DI.10
		END_MACRO
		#593 MACRO 8 bit output module 3()
			#594 panStartN010501 <= N0105statStartedP1
			#595 panStartN010502 <= N0105statStartedP2
			#596 panCleanFS020101 <= DD6_DI.20
			#597 panCleanFS020102 <= DD6_DI.22
			#598 panCleanFS020103 <= DD6_DI.24
			#599 panCleanFS020104 <= DD6_DI.26
			#600 panCleanFS020105 <= DD6_DI.28
			#601 panCleanFS020106 <= DD6_DI.30
		END_MACRO
		#602 MACRO 8 bit output module 4()
			#603 panCleanFS020201 <= DD7_DI. 0
			#604 panCleanFS020202 <= DD7_DI. 2
			#605 panCleanFS020203 <= DD7_DI. 4
			#606 panCleanFS020204 <= DD7_DI. 6
			#607 panCleanFS020205 <= DD7_DI. 8
			#608 panCleanFS020206 <= DD7_DI. 10
			#609 panSludgeReady <= DD7_DI.15
			#610 panStartN0401 <= DD7_DI.13
		END_MACRO
		#611 MACRO 8 bit output module 5()
			#612 panKSHE0401open <= DD9_DI.2
			#613 panFPKready <= DD7_DI.12
			#614 panFPKneedToClean <= FPKneedToClean
			#615 panStartN040401 <= DD5_DI.16
			#616 panStartN040402 <= DD5_DI.17
			#617 panStartUFO030101 <= DD5_DI.26
			#618 panStartUFO030102 <= DD5_DI.28
			#619 panAlarm <= alarm
		END_MACRO
		#620 MACRO 8 bit output module 6()
			#621 panErrorTempSensor <= DD1_AI0_error
			#622 panErrorFT0101 <= DD1_AI1_error
			#623 panErrorFT0102 <= DD1_AI2_error
			#624 panErrorQE0102 <= DD1_AI3_error
			#625 panErrorQE0102 <= DD1_AI4_error
			#626 panAlarmHighTemp <= alarmHighTemperature
			#627 panAlarmLowTemp <= alarmLowTemperature
			#628 panND0502dosingError <= ND0502dosingError
		END_MACRO
		#629 MACRO 8 bit output module 7()
			#630 panND0602dosingError <= ND0602dosingError
			#631 panND0603dosingError <= ND0603dosingError
			#632 panND0803dosingError <= ND0803dosingError
			#633 panND0804dosingError <= ND0804dosingError
			#634 panND080301emptyAlarm <= DD1_DI6
			#635 panND080302emptyAlarm <= DD1_DI7
			#636 panN010501alarm <= N010501alarm
			#637 panN010502alarm <= N010502alarm
		END_MACRO
		#638 MACRO 8 bit output module 8()
			#639 panZDE0225errorToOpen <= ZDE0225errorToOpen
			#640 panZDE0225errorToClose <= ZDE0225errorToClose
			#641 panFPKalarm <= DD7_DI.14
			#642 panFPKnotStarted <= FPKnotStarted
			#643 panErrorFPKsensor <= DD1_AI5_error
			#644 panFPKkshe0401errorToOpen <= FPKkshe0401errorToOpen
			#645 panFPKkshe0401errorToClose <= FPKkshe0401errorToClose
			#646 panUFO030101alarm <= DD5_DI.27
		END_MACRO
		#647 MACRO 8 bit output module 9()
			#648 panUFO030102alarm <= DD5_DI.29
			#649 panFilterFailToRegen020101 <= filterFailToRegen020101
			#650 panErrorToOpenZD0201 <= errorToOpenZD0201
			#651 panErrorToCloseZD0201 <= errorToCloseZD0201
			#652 panErrorToOpenZD0207 <= errorToOpenZD0207
			#653 panErrorToCloseZD0207 <= errorToCloseZD0207
			#654 panFilterFailToRegen020102 <= filterFailToRegen020102
			#655 panErrorToOpenZD0202 <= errorToOpenZD0202
		END_MACRO
		#656 MACRO 8 bit output module 10()
			#657 panErrorToCloseZD0202 <= errorToCloseZD0202
			#658 panErrorToOpenZD0208 <= errorToOpenZD0208
			#659 panErrorToCloseZD0208 <= errorToCloseZD0208
			#660 panFilterFailToRegen020103 <= filterFailToRegen020103
			#661 panErrorToOpenZD0203 <= errorToOpenZD0203
			#662 panErrorToCloseZD0203 <= errorToCloseZD0203
			#663 panErrorToOpenZD0209 <= errorToOpenZD0209
			#664 panErrorToCloseZD0209 <= errorToCloseZD0209
		END_MACRO
		#665 MACRO 8 bit output module 11()
			#666 panFilterFailToRegen020104 <= filterFailToRegen020104
			#667 panErrorToOpenZD0204 <= errorToOpenZD0204
			#668 panErrorToCloseZD0204 <= errorToCloseZD0204
			#669 panErrorToOpenZD0210 <= errorToOpenZD0210
			#670 panErrorToCloseZD0210 <= errorToCloseZD0210
			#671 panFilterFailToRegen020105 <= filterFailToRegen020105
			#672 panErrorToOpenZD0205 <= errorToOpenZD0205
			#673 panErrorToCloseZD0205 <= errorToCloseZD0205
		END_MACRO
		#674 MACRO 8 bit output module 12()
			#675 panErrorToOpenZD0211 <= errorToOpenZD0211
			#676 panErrorToCloseZD0211 <= errorToCloseZD0211
			#677 panFilterFailToRegen020106 <= filterFailToRegen020106
			#678 panErrorToOpenZD0206 <= errorToOpenZD0206
			#679 panErrorToCloseZD0206 <= errorToCloseZD0206
			#680 panErrorToOpenZD0212 <= errorToOpenZD0212
			#681 panErrorToCloseZD0212 <= errorToCloseZD0212
			#682 panFilterFailToRegen020201 <= filterFailToRegen020201
		END_MACRO
		#683 MACRO 8 bit output module 13()
			#684 panErrorToOpenZD0213 <= errorToOpenZD0213
			#685 panErrorToCloseZD0213 <= errorToCloseZD0213
			#686 panErrorToOpenZD0219 <= errorToOpenZD0219
			#687 panErrorToCloseZD0219 <= errorToCloseZD0219
			#688 panFilterFailToRegen020202 <= filterFailToRegen020202
			#689 panErrorToOpenZD0214 <= errorToOpenZD0214
			#690 panErrorToCloseZD0214 <= errorToCloseZD0214
			#691 panErrorToOpenZD0220 <= errorToOpenZD0220
		END_MACRO
		#692 MACRO 8 bit output module 14()
			#693 panErrorToCloseZD0220 <= errorToCloseZD0220
			#694 panFilterFailToRegen020203 <= filterFailToRegen020203
			#695 panErrorToOpenZD0215 <= errorToOpenZD0215
			#696 panErrorToCloseZD0215 <= errorToCloseZD0215
			#697 panErrorToOpenZD0221 <= errorToOpenZD0221
			#698 panErrorToCloseZD0221 <= errorToCloseZD0221
			#699 panFilterFailToRegen020204 <= filterFailToRegen020204
			#700 panErrorToOpenZD0216 <= errorToOpenZD0216
		END_MACRO
		#701 MACRO 8 bit output module 15()
			#702 panErrorToCloseZD0216 <= errorToCloseZD0216
			#703 panErrorToOpenZD0222 <= errorToOpenZD0222
			#704 panErrorToCloseZD0222 <= errorToCloseZD0222
			#705 panFilterFailToRegen020205 <= filterFailToRegen020205
			#706 panErrorToOpenZD0217 <= errorToOpenZD0217
			#707 panErrorToCloseZD0217 <= errorToCloseZD0217
			#708 panErrorToOpenZD0223 <= errorToOpenZD0223
			#709 panErrorToCloseZD0223 <= errorToCloseZD0223
		END_MACRO
		#710 MACRO 8 bit output module 16()
			#711 panFilterFailToRegen020206 <= filterFailToRegen020206
			#712 panErrorToOpenZD0218 <= errorToOpenZD0218
			#713 panErrorToCloseZD0218 <= errorToCloseZD0218
			#714 panErrorToOpenZD0224 <= errorToOpenZD0224
			#715 panErrorToCloseZD0224 <= errorToCloseZD0224
			#716 panAlarmPLKnetwork <= alarmPLKnetwork
			#717 panAlarmND050201 <= alarmND050201
			#718 panAlarmND050202 <= alarmND050202
		END_MACRO
		#719 MACRO 8 bit output module 17()
			#720 panAlarmND060201 <= alarmND060201
			#721 panAlarmND060202 <= alarmND060202
			#722 panAlarmND060301 <= alarmND060301
			#723 panAlarmND060302 <= alarmND060302
			#724 panAlarmND070301 <= alarmND070301
			#725 panAlarmND070302 <= alarmND070302
			#726 panAlarmND080301 <= alarmND080301
			#727 panAlarmND080302 <= alarmND080302
		END_MACRO
		#728 MACRO 8 bit output module 18()
			#729 panAlarmND0804 <= alarmND0804
			#730 panAlarmOGM0104overload <= alarmOGM0104overload
			#731 panAlarmRCHV0203overload <= alarmRCHV0203overload
			#732 panAlarmN040402 <= alarmN040402
			#733 panAlarmN040401 <= alarmN040401
			#734 panAlarmM0604 <= alarmM0604
			#735 panAlarmM0702 <= alarmM0702
			#736 panAlarmM0802 <= alarmM0802
		END_MACRO
		#737 MACRO 8 bit output module 19()
			#738 panAlarmN020401 <= alarmN020401
			#739 panAlarmN020402 <= alarmN020402
			#740 panAlarmFS020101 <= alarmFS020101
			#741 panAlarmFS020102 <= alarmFS020102
			#742 panAlarmFS020103 <= alarmFS020103
			#743 panAlarmFS020104 <= alarmFS020104
			#744 panAlarmFS020105 <= alarmFS020105
			#745 panAlarmFS020106 <= alarmFS020106
		END_MACRO
		#746 MACRO 8 bit output module 20()
			#747 panAlarmFS020201 <= alarmFS020201
			#748 panAlarmFS020202 <= alarmFS020202
			#749 panAlarmFS020203 <= alarmFS020203
			#750 panAlarmFS020204 <= alarmFS020204
			#751 panAlarmFS020205 <= alarmFS020205
			#752 panAlarmFS020206 <= alarmFS020206
			#753 panAlarmZDE0201power <= alarmZDE0201power
			#754 panAlarmZDE0202power <= alarmZDE0202power
		END_MACRO
		#755 MACRO 8 bit output module 21()
			#756 panAlarmZDE0203power <= alarmZDE0203power
			#757 panAlarmZDE0204power <= alarmZDE0204power
			#758 panAlarmZDE0205power <= alarmZDE0205power
			#759 panAlarmZDE0206power <= alarmZDE0206power
			#760 panAlarmZDE0207power <= alarmZDE0207power
			#761 panAlarmZDE0208power <= alarmZDE0208power
			#762 panAlarmZDE0209power <= alarmZDE0209power
			#763 panAlarmZDE0210power <= alarmZDE0210power
		END_MACRO
		#764 MACRO 8 bit output module 22()
			#765 panAlarmZDE0211power <= alarmZDE0211power
			#766 panAlarmZDE0212power <= alarmZDE0212power
			#767 panAlarmZDE0213power <= alarmZDE0213power
			#768 panAlarmZDE0214power <= alarmZDE0214power
			#769 panAlarmZDE0215power <= alarmZDE0215power
			#770 panAlarmZDE0216power <= alarmZDE0216power
			#771 panAlarmZDE0217power <= alarmZDE0217power
			#772 panAlarmZDE0218power <= alarmZDE0218power
		END_MACRO
		#773 MACRO 8 bit output module 23()
			#774 panAlarmZDE0219power <= alarmZDE0219power
			#775 panAlarmZDE0220power <= alarmZDE0220power
			#776 panAlarmZDE0221power <= alarmZDE0221power
			#777 panAlarmZDE0222power <= alarmZDE0222power
			#778 panAlarmZDE0223power <= alarmZDE0223power
			#779 panAlarmZDE0224power <= alarmZDE0224power
			#780 panAlarmZDE0225power <= alarmZDE0225power
			#781 panAlarmKSHE0401power <= alarmKSHE0401power
		END_MACRO
		#782 MACRO 8 bit output module 24()
			#783 panAlarmKNS <= alarmKNS
			#784 panAlarmPowerSocketFS <= alarmPowerSocketFS
			#785 panAlarmKEMvalvesPower <= alarmKEMvalvesPower
			#786 panAlarmEmergencyPressed <= alarmEmergencyPressed
			#787 panAlarmRKF <= alarmRKF
			#788 panUFO0301noFlowAttention <= UFO0301noFlowAttention
			#789 panM0604attention <= M0604attention
			#790 panM0702attention <= M0702attention
		END_MACRO
		#791 MACRO 8 bit output module 25()
			#792 panM0802attention <= M0802attention
			#793 panStatusKNS <= DD6_DI.8
			#794 panND0502statRegimeP1M <= ND0502statRegimeP1M
			#795 panND0502statRegimeP2M <= ND0502statRegimeP2M
			#796 panND0502statRegimeByC <= ND0502statRegimeByC
			#797 panND0502statRegimeByWT <= ND0502statRegimeByWT
			#798 panND0602statRegimeP1M <= ND0602statRegimeP1M
			#799 panND0602statRegimeP2M <= ND0602statRegimeP2M
		END_MACRO
		#800 MACRO 8 bit output module 26()
			#801 panND0602statRegimeByC <= ND0602statRegimeByC
			#802 panND0602statRegimeByWT <= ND0602statRegimeByWT
			#803 panND0603statRegimeP1M <= ND0603statRegimeP1M
			#804 panND0603statRegimeP2M <= ND0603statRegimeP2M
			#805 panND0603statRegimeByC <= ND0603statRegimeByC
			#806 panND0603statRegimeByWT <= ND0603statRegimeByWT
			#807 panND0703statRegimeP1M <= ND0703statRegimeP1M
			#808 panND0703statRegimeP2M <= ND0703statRegimeP2M
		END_MACRO
		#809 MACRO 8 bit output module 27()
			#810 panND0703statRegimeByC <= ND0703statRegimeByC
			#811 panND0703statRegimeByWT <= ND0703statRegimeByWT
			#812 panND0803statRegimeP1M <= ND0803statRegimeP1M
			#813 panND0803statRegimeP2M <= ND0803statRegimeP2M
			#814 panND0803statRegimeByC <= ND0803statRegimeByC
			#815 panND0803statRegimeByWT <= ND0803statRegimeByWT
			#816 panN0105statRegimeP1M <= N0105statRegimeP1M
			#817 panN0105statRegimeP2M <= N0105statRegimeP2M
		END_MACRO
		#818 MACRO 8 bit output module 28()
			#819 panN0105statRegimeByC <= N0105statRegimeByC
			#820 panN0105statRegimeByWT <= N0105statRegimeByWT
			#821 panN0204statRegimeP1M <= N0204statRegimeP1M
			#822 panN0204statRegimeP2M <= N0204statRegimeP2M
			#823 panN0204statRegimeByC <= N0204statRegimeByC
			#824 panN0204statRegimeWT <= N0204statRegimeWT
			#825 panN0404statRegimeP1M <= N0404statRegimeP1M
			#826 panN0404statRegimeP2M <= N0404statRegimeP2M
		END_MACRO
		#827 MACRO 8 bit output module 29()
			#828 panN0404statRegimeByC <= N0404statRegimeByC
			#829 panN0404statRegimeWT <= N0404statRegimeWT
			#830 panUFO0301statRegimeP1M <= UFO0301statRegimeP1M
			#831 panUFO0301statRegimeP2M <= UFO0301statRegimeP2M
			#832 panUFO0301statRegimeByC <= UFO0301statRegimeByC
			#833 panUFO0301statRegimeWT <= UFO0301statRegimeWT
			#834 panZDE0225open <= DD9_DI.0
			#835 panZDE0201open <= DD7_DI.16
		END_MACRO
		#836 MACRO 8 bit output module 30()
			#837 panZDE0201close <= DD7_DI.17
			#838 panZDE0202open <= DD7_DI.18
			#839 panZDE0202close <= DD7_DI.19
			#840 panZDE0203open <= DD7_DI.20
			#841 panZDE0203close <= DD7_DI.21
			#842 panZDE0204open <= DD7_DI.22
			#843 panZDE0204close <= DD7_DI.23
			#844 panZDE0205open <= DD7_DI.24
		END_MACRO
		#845 MACRO 8 bit output module 31()
			#846 panZDE0205close <= DD7_DI.25
			#847 panZDE0206open <= DD7_DI.26
			#848 panZDE0206close <= DD7_DI.27
			#849 panZDE0207open <= DD7_DI.28
			#850 panZDE0207close <= DD7_DI.29
			#851 panZDE0208open <= DD7_DI.30
			#852 panZDE0208close <= DD7_DI.31
			#853 panZDE0209open <= DD8_DI.0
		END_MACRO
		#854 MACRO 8 bit output module 32()
			#855 panZDE0209close <= DD8_DI.1
			#856 panZDE0210open <= DD8_DI.2
			#857 panZDE0210close <= DD8_DI.3
			#858 panZDE0211open <= DD8_DI.4
			#859 panZDE0211close <= DD8_DI.5
			#860 panZDE0212open <= DD8_DI.6
			#861 panZDE0212close <= DD8_DI.7
			#862 panZDE0213open <= DD8_DI.8
		END_MACRO
		#863 MACRO 8 bit output module 33()
			#864 panZDE0213close <= DD8_DI.9
			#865 panZDE0214open <= DD8_DI.10
			#866 panZDE0214close <= DD8_DI.11
			#867 panZDE0215open <= DD8_DI.12
			#868 panZDE0215close <= DD8_DI.13
			#869 panZDE0216open <= DD8_DI.14
			#870 panZDE0216close <= DD8_DI.15
			#871 panZDE0217open <= DD8_DI.16
		END_MACRO
		#872 MACRO 8 bit output module 34()
			#873 panZDE0217close <= DD8_DI.17
			#874 panZDE0218open <= DD8_DI.18
			#875 panZDE0218close <= DD8_DI.19
			#876 panZDE0219open <= DD8_DI.20
			#877 panZDE0219close <= DD8_DI.21
			#878 panZDE0220open <= DD8_DI.22
			#879 panZDE0220close <= DD8_DI.23
			#880 panZDE0221open <= DD8_DI.24
		END_MACRO
		#881 MACRO 8 bit output module 35()
			#882 panZDE0221close <= DD8_DI.25
			#883 panZDE0222open <= DD8_DI.26
			#884 panZDE0222close <= DD8_DI.27
			#885 panZDE0223open <= DD8_DI.28
			#886 panZDE0223close <= DD8_DI.29
			#887 panZDE0224open <= DD8_DI.30
			#888 panZDE0224close <= DD8_DI.31
			#889 panZDE0225close <= DD9_DI.1
		END_MACRO
		#890 MACRO 8 bit output module 36x()
			#891 panKSHE0401close <= DD9_DI.3
			#892 panZDE0301open <= DD1_DI12
			#893 panZDE0301close <= DD1_DI13
			#894 panZDE0302open <= DD1_DI14
			#895 panZDE0302close <= DD1_DI15
			#896 panErrorToOpenZDE0301 <= errorToOpenZDE0301
			#897 panErrorToCloseZDE0301 <= errorToCloseZDE0301
			#898 panErrorToOpenZDE0302 <= errorToOpenZDE0302
		END_MACRO
		#899 panErrorToCloseZDE0302 <= errorToCloseZDE0302
		#900 panAlarmZDE0301power <= alarmZDE0301power
		#901 panAlarmZDE0302power <= alarmZDE0302power
	END_MACRO
	#902 MACRO PFW регистры на чтение из панели (управление ПЛК)()
		#903 MUL(panTimeToOpenCloseValve, 1000)
		#904 REAL_TO_TIME(#903)
		#905 TimeToOpenCloseValve <= #904
		#906 maxTemperature <= panMaxTemperature
		#907 minTemperature <= panMinTemperature
		#908 ND0502setMaxDosVal <= panND0502setMaxDosVal
		#909 ND0502setKoefProp <= panND0502setKoefProp
		#910 ND0602setMaxDosVal <= panND0602setMaxDosVal
		#911 ND0602setKoefProp <= panND0602setKoefProp
		#912 ND0603setMaxDosVal <= panND0603setMaxDosVal
		#913 ND0603setKoefProp <= panND0603setKoefProp
		#914 ND0703pHsetValue <= panND0703pHsetValue
		#915 ND0703YoutManual <= panND0703YoutManual
		#916 ND0703koeffI <= panND0703koeffI
		#917 ND0703koeffD <= panND0703koeffD
		#918 ND0703koeffP <= panND0703koeffP
		#919 ND0803setMaxDosVal <= panND0803setMaxDosVal
		#920 ND0803setKoefProp <= panND0803setKoefProp
		#921 ND0804doseValue <= panND0804doseValue
		#922 N0105flowSetValue <= panN0105flowSetValue
		#923 N0105YoutManual <= panN0105YoutManual
		#924 N0105koeffI <= panN0105koeffI
		#925 N0105koeffD <= panN0105koeffD
		#926 N0105koeffP <= panN0105koeffP
		#927 FQS0301impulsValue <= panFQS0301impulsValue
		#928 FQS0301correction <= panFQS0301correction
		#929 MUL(panFPKtimeToWork, 1000)
		#930 REAL_TO_TIME(#929)
		#931 FPKtimeToWork <= #930
		#932 MUL(panFPKnotStartedTime, 1000)
		#933 REAL_TO_TIME(#932)
		#934 FPKnotStartedTime <= #933
		#935 FPKmaxPressureValue <= panFPKmaxPressureValue
		#936 filterValueToRegen <= panFilterValueToRegen
	END_MACRO
	#937 MACRO PSB регистры на чтение из панели (управление ПЛК)()
		(* PSB регистры на чтение из панели (управление ПЛК) *)
		#938 MACRO 8 bit input module 1()
			#939 alarmReset <= panAlarmResetButton
			#940 ND0502resetCountP1 <= panND0502resetCountP1
			#941 ND0502resetCountP2 <= panND0502resetCountP2
			#942 ND0502resetWorkTimeP1 <= panND0502resetWorkTimeP1
			#943 ND0502resetWorkTimeP2 <= panND0502resetWorkTimeP2
			#944 ND0502regimeP1M <= panND0502regimeP1M
			#945 ND0502regimeP2M <= panND0502regimeP2M
			#946 ND0502regimeByC <= panND0502regimeByC
		END_MACRO
		#947 MACRO 8 bit input module 2()
			#948 ND0502regimeByWT <= panND0502regimeByWT
			#949 ND0602resetCountP1 <= panND0602resetCountP1
			#950 ND0602resetCountP2 <= panND0602resetCountP2
			#951 ND0602resetWorkTimeP1 <= panND0602resetWorkTimeP1
			#952 ND0602resetWorkTimeP2 <= panND0602resetWorkTimeP2
			#953 ND0602regimeP1M <= panND0602regimeP1M
			#954 ND0602regimeP2M <= panND0602regimeP2M
			#955 ND0602regimeByC <= panND0602regimeByC
		END_MACRO
		#956 MACRO 8 bit input module 3()
			#957 ND0602regimeByWT <= panND0602regimeByWT
			#958 ND0603resetCountP1 <= panND0603resetCountP1
			#959 ND0603resetCountP2 <= panND0603resetCountP2
			#960 ND0603resetWorkTimeP1 <= panND0603resetWorkTimeP1
			#961 ND0603resetWorkTimeP2 <= panND0603resetWorkTimeP2
			#962 ND0603regimeP1M <= panND0603regimeP1M
			#963 ND0603regimeP2M <= panND0603regimeP2M
			#964 ND0603regimeByC <= panND0603regimeByC
		END_MACRO
		#965 MACRO 8 bit input module 4()
			#966 ND0603regimeByWT <= panND0603regimeByWT
			#967 ND0703resetCountP1 <= panND0703resetCountP1
			#968 ND0703resetCountP2 <= panND0703resetCountP2
			#969 ND0703resetWorkTimeP1 <= panND0703resetWorkTimeP1
			#970 ND0703resetWorkTimeP2 <= panND0703resetWorkTimeP2
			#971 ND0703regimeP1M <= panND0703regimeP1M
			#972 ND0703regimeP2M <= panND0703regimeP2M
			#973 ND0703regimeByC <= panND0703regimeByC
		END_MACRO
		#974 MACRO 8 bit input module 5()
			#975 ND0703regimeByWT <= panND0703regimeByWT
			#976 ND0703YmanAuto <= panND0703YmanAuto
			#977 ND0803resetCountP1 <= panND0803resetCountP1
			#978 ND0803resetCountP2 <= panND0803resetCountP2
			#979 ND0803resetWorkTimeP1 <= panND0803resetWorkTimeP1
			#980 ND0803resetWorkTimeP2 <= panND0803resetWorkTimeP2
			#981 ND0803regimeP1M <= panND0803regimeP1M
			#982 ND0803regimeP2M <= panND0803regimeP2M
		END_MACRO
		#983 MACRO 8 bit input module 6()
			#984 ND0803regimeByC <= panND0803regimeByC
			#985 ND0803regimeByWT <= panND0803regimeByWT
			#986 N0105resetCountP1 <= panN0105resetCountP1
			#987 N0105resetCountP2 <= panN0105resetCountP2
			#988 N0105resetWorkTimeP1 <= panN0105resetWorkTimeP1
			#989 N0105resetWorkTimeP2 <= panN0105resetWorkTimeP2
			#990 N0105regimeByC <= panN0105regimeByC
			#991 N0105regimeByWT <= panN0105regimeByWT
		END_MACRO
		#992 MACRO 8 bit input module 7()
			#993 N0105YmanAuto <= panN0105YmanAuto
			#994 N0204resetCountP1 <= panN0204resetCountP1
			#995 N0204resetCountP2 <= panN0204resetCountP2
			#996 N0204resetWorkTimeP1 <= panN0204resetWorkTimeP1
			#997 N0204resetWorkTimeP2 <= panN0204resetWorkTimeP2
			#998 N0204regimeP1M <= panN0204regimeP1M
			#999 N0204regimeP2M <= panN0204regimeP2M
			#1000 N0204regimeByC <= panN0204regimeByC
		END_MACRO
		#1001 MACRO 8 bit input module 8()
			#1002 N0204regimeWT <= panN0204regimeWT
			#1003 UFO0301resetCountP1 <= panUFO0301resetCountP1
			#1004 UFO0301resetCountP2 <= panUFO0301resetCountP2
			#1005 UFO0301resetWorkTimeP1 <= panUFO0301resetWorkTimeP1
			#1006 UFO0301resetWorkTimeP2 <= panUFO0301resetWorkTimeP2
			#1007 UFO0301regimeP1M <= panUFO0301regimeP1M
			#1008 UFO0301regimeP2M <= panUFO0301regimeP2M
			#1009 UFO0301regimeByC <= panUFO0301regimeByC
		END_MACRO
		#1010 MACRO 8 bit input module 9()
			#1011 UFO0301regimeWT <= panUFO0301regimeWT
			#1012 N0404resetCountP1 <= panN0404resetCountP1
			#1013 N0404resetCountP2 <= panN0404resetCountP2
			#1014 N0404resetWorkTimeP1 <= panN0404resetWorkTimeP1
			#1015 N0404resetWorkTimeP2 <= panN0404resetWorkTimeP2
			#1016 N0404regimeP1M <= panN0404regimeP1M
			#1017 N0404regimeP2M <= panN0404regimeP2M
			#1018 N0404regimeByC <= panN0404regimeByC
		END_MACRO
		#1019 MACRO 8 bit input module 10-11()
			(* одули 10 и 11 заполнены переменными для тестирования задвижек. / Здесь они не показаны, т.к. спешка. / Они вставлены напрямую в макросы управления промывкой фильтров. / testValvesFS020101 - testValvesFS020206 (PSB612-623) *)
			#1020 N0404regimeWT <= panN0404regimeWT
			#1021 FQS0301reset <= panFQS0301reset
			#1022 FQS0301addCorrection <= panFQS0301addCorrection
			#1023 FQS0301deleteCorrection <= panFQS0301deleteCorrection
		END_MACRO
		#1024 testKSHE0401 <= panTestKSHE0401
		#1025 testZDE0225 <= panTestZDE0225
		#1026 testZDE03 <= panTestZDE03
		#1027 manualZDE0301 <= panManualZDE0301
		#1028 manualZDE0302 <= panManualZDE0302
	END_MACRO
END_MACRO
#1029 NOT(DD6_DI.13)
#1030 alarmRCHV0203overload <= #1029
#1031 NOT(DD9_DI.5)
#1032 alarmZDE0202power <= #1031
#1033 NOT(DD9_DI.26)
#1034 alarmZDE0223power <= #1033
#1035 MACRO переменные на диспетчеризацию()
	#1036 remFT0101value <= DD1_AI1_FT0101value
	#1037 remFQS0301totalAmount <= FQS0301totalAmount
	#1038 remTemperatureValue <= temperatureValue
	#1039 remStatusN010501started <= N0105statStartedP1
	#1040 remStatusN010502started <= N0105statStartedP2
	#1041 remStatusUFO030101started <= DD5_DI.26
	#1042 remStatusUFO030102started <= DD5_DI.28
	#1043 remAlarm <= Alarm
	#1044 remN010501alarm <= N010501alarm
	#1045 remN010502alarm <= N010502alarm
	#1046 remFPKalarm <= DD7_DI.14
	#1047 remUFO030101alarm <= DD5_DI.27
	#1048 remUFO030102alarm <= DD5_DI.29
	#1049 remAlarmEmergencyPressed <= alarmEmergencyPressed
	#1050 remAlarmOOGM0104overload <= DD6_DI.11
	#1051 remAlarmRCHV0203overload <= DD6_DI.13
END_MACRO
#1052 NOT(DD5_DI.14)
#1053 alarmN040402 <= #1052
#1054 NOT(DD9_DI.6)
#1055 alarmZDE0203power <= #1054
#1056 NOT(DD9_DI.27)
#1057 alarmZDE0224power <= #1056
#1058 NOT(DD5_DI.15)
#1059 alarmN040401 <= #1058
#1060 NOT(DD9_DI.7)
#1061 alarmZDE0204power <= #1060
#1062 NOT(DD9_DI.28)
#1063 alarmZDE0225power <= #1062
#1064 NOT(DD5_DI.20)
#1065 alarmM0604 <= #1064
#1066 NOT(DD9_DI.8)
#1067 alarmZDE0205power <= #1066
#1068 NOT(DD9_DI.29)
#1069 alarmKSHE0401power <= #1068
#1070 NOT(DD5_DI.22)
#1071 alarmM0702 <= #1070
#1072 NOT(DD9_DI.9)
#1073 alarmZDE0206power <= #1072
#1074 NOT(DD6_DI.9)
#1075 alarmKNS <= #1074
#1076 NOT(DD5_DI.24)
#1077 alarmM0802 <= #1076
#1078 NOT(DD9_DI.10)
#1079 alarmZDE0207power <= #1078
#1080 NOT(DD6_DI.17)
#1081 alarmPowerSocketFS <= #1080
#1082 NOT(DD5_DI.7)
#1083 alarmN020401 <= #1082
#1084 NOT(DD9_DI.11)
#1085 alarmZDE0208power <= #1084
#1086 NOT(DD6_DI.18)
#1087 alarmKEMvalvesPower <= #1086
#1088 NOT(DD5_DI.8)
#1089 alarmN020402 <= #1088
#1090 NOT(DD9_DI.12)
#1091 alarmZDE0209power <= #1090
#1092 NOT(DD1_DI4)
#1093 alarmEmergencyPressed <= #1092
#1094 GT(DD1_AI2_FT0102value, 0)
#1095 filterPulserGen:PulsePerSec(start: #1094)
#1096 DIV(DD1_AI2_FT0102value, 3600)
#1097 ADD(EN: #1095.out, #1096, filterTotalAmountFT0102)
#1098 filterTotalAmountFT0102 <= #1097
#1099 NOT(DD6_DI.21)
#1100 alarmFS020101 <= #1099
#1101 NOT(DD9_DI.13)
#1102 alarmZDE0210power <= #1101
#1103 NOT(DD1_DI5)
#1104 alarmRKF <= #1103
#1105 NOT(DD9_DI.30)
#1106 alarmZDE0301power <= #1105
#1107 NOT(DD9_DI.31)
#1108 alarmZDE0302power <= #1107
#1109 MOVE(EN: filterTotalAmountReset, 0)
#1110 filterTotalAmountFT0102 <= #1109
#1111 GE(filterTotalAmountFT0102, filterValueToRegen)
#1112 MACRO управление промывкой фильтра ФС02.01.01(pin 1 "сигнал на промывку": #1111, pin 2 "авария фильтра": DD6_DI.21, pin 3 "подтверждение промывки": DD6_DI.20, pin 4 "сброс аварий": alarmReset, pin 5 "начать очередь снова": filterStartNewQueue, pin 6 "ЗДЭ02.01 открыта": DD7_DI.16, pin 7 "ЗДЭ02.01 закрыта": DD7_DI.17, pin 8 "ЗДЭ02.07 открыта": DD7_DI.28, pin 9 "ЗДЭ02.07 закрыта": DD7_DI.29, pin 10 "время движения ЗДЭ": timeToOpenCloseValve, pin 11 "авария питания ЗДЭ02.01": DD9_DI.4, pin 12 "авария питания ЗДЭ02.07": DD9_DI.10)
	(* <- выход использовать в / последнем фильтре для / начала очереди заново *)
	(* если открыт = промывка *)
	(* если открыт = фильтрация *)
	out 1 "следующий в очереди" <= #1115.output
	out 2 "промыть ФС02.01.01" <= #1114
	#1113 ZD0201:SimpleValve(inputOpen: NOT #1114, inputClose: #1114, statusOpen: pin 6, statusClose: pin 7, reset: pin 4, timeToOpenClose: pin 10)
	out 6 "открыть ЗДЭ02.01" <= #1113.outputOpen
	out 7 "закрыть ЗДЭ02.01" <= #1113.outputClose
	out 8 "авария открытия ЗДЭ02.01" <= #1113.errorToOpen
	#1114 OR(panTestValvesFS020101, #1115.regenFilterOUT)
	out 9 "авария закрытия ЗДЭ02.01" <= #1113.errorToClose
	#1115 FS020101manager:FilterQueueManager(input: pin 1, filterAlarm: #1116, regenFilterStatus: pin 3, alarmReset: pin 4, startNextLoop: pin 5)
	#1116 OR(alarmZD020107, pin 2, pin 11, pin 12)
	out 3 "ФС02.01.01 промыт" <= #1115.regenerated
	out 4 "не удалось промыть" <= #1115.failToRegen
	#1117 OR(#1113.errorToOpen, #1113.errorToClose, #1119.errorToOpen, #1119.errorToClose)
	#1118 alarmZD020107 <= #1117
	out 5 "сброс счетчика" <= #1115.counterReset
	#1119 ZD0207:SimpleValve(inputOpen: #1114, inputClose: NOT #1114, statusOpen: pin 8, statusClose: pin 9, reset: pin 4, timeToOpenClose: pin 10)
	out 10 "открыть ЗДЭ02.07" <= #1119.outputOpen
	out 11 "закрыть ЗДЭ02.07" <= #1119.outputClose
	out 12 "авария открытия ЗДЭ02.07" <= #1119.errorToOpen
	out 13 "авария закрытия ЗДЭ02.07" <= #1119.errorToClose
END_MACRO
#1120 DD2_DO.4 <= #1112.out 2
#1121 regeneratedFS020101 <= #1112.out 3
#1122 filterFailToRegen020101 <= #1112.out 4
#1123 filterTotalAmountReset <= #1112.out 5
#1124 DD2_DO.16 <= #1112.out 6
#1125 DD2_DO.17 <= #1112.out 7
#1126 errorToOpenZD0201 <= #1112.out 8
#1127 errorToCloseZD0201 <= #1112.out 9
#1128 DD2_DO.28 <= #1112.out 10
#1129 DD2_DO.29 <= #1112.out 11
#1130 errorToOpenZD0207 <= #1112.out 12
#1131 errorToCloseZD0207 <= #1112.out 13
#1132 MACRO управление промывкой фильтра ФС02.01.02(pin 1 "сигнал на промывку": #1112.out 1, pin 2 "авария фильтра": DD6_DI.23, pin 3 "подтверждение промывки": DD6_DI.22, pin 4 "сброс аварий": alarmReset, pin 5 "начать очередь снова": filterStartNewQueue, pin 6 "ЗДЭ02.02 открыта": DD7_DI.18, pin 7 "ЗДЭ02.02 закрыта": DD7_DI.19, pin 8 "ЗДЭ02.08 открыта": DD7_DI.30, pin 9 "ЗДЭ02.08 закрыта": DD7_DI.31, pin 10 "время движения ЗДЭ": timeToOpenCloseValve, pin 11 "авария питания ЗДЭ02.02": DD9_DI.5, pin 12 "авария питания ЗДЭ02.08": DD9_DI.11)
	(* <- выход использовать в / последнем фильтре для / начала очереди заново *)
	(* если открыт = промывка *)
	(* если открыт = фильтрация *)
	out 1 "следующий в очереди" <= #1135.output
	out 2 "промыть ФС02.01.02" <= #1134
	#1133 ZD0202:SimpleValve(inputOpen: NOT #1134, inputClose: #1134, statusOpen: pin 6, statusClose: pin 7, reset: pin 4, timeToOpenClose: pin 10)
	out 5 "открыть ЗДЭ02.02" <= #1133.outputOpen
	out 6 "закрыть ЗДЭ02.02" <= #1133.outputClose
	out 7 "авария открытия ЗДЭ02.02" <= #1133.errorToOpen
	#1134 OR(panTestValvesFS020102, #1135.regenFilterOUT)
	out 8 "авария закрытия ЗДЭ02.02" <= #1133.errorToClose
	#1135 FS020102manager:FilterQueueManager(input: pin 1, filterAlarm: #1136, regenFilterStatus: pin 3, alarmReset: pin 4, startNextLoop: pin 5)
	#1136 OR(alarmZD020208, pin 2, pin 11, pin 12)
	#1137 OR(#1133.errorToOpen, #1133.errorToClose, #1139.errorToOpen, #1139.errorToClose)
	#1138 alarmZD020208 <= #1137
	out 3 "ФС02.01.02 промыт" <= #1135.regenerated
	out 4 "не удалось промыть" <= #1135.failToRegen
	#1139 ZD0208:SimpleValve(inputOpen: #1134, inputClose: NOT #1134, statusOpen: pin 8, statusClose: pin 9, reset: pin 4, timeToOpenClose: pin 10)
	out 9 "открыть ЗДЭ02.08" <= #1139.outputOpen
	out 10 "закрыть ЗДЭ02.08" <= #1139.outputClose
	out 11 "авария открытия ЗДЭ02.08" <= #1139.errorToOpen
	out 12 "авария закрытия ЗДЭ02.08" <= #1139.errorToClose
END_MACRO
#1140 DD2_DO.5 <= #1132.out 2
#1141 regeneratedFS020102 <= #1132.out 3
#1142 filterFailToRegen020102 <= #1132.out 4
#1143 DD2_DO.18 <= #1132.out 5
#1144 DD2_DO.19 <= #1132.out 6
#1145 errorToOpenZD0202 <= #1132.out 7
#1146 errorToCloseZD0202 <= #1132.out 8
#1147 DD2_DO.30 <= #1132.out 9
#1148 DD2_DO.31 <= #1132.out 10
#1149 errorToOpenZD0208 <= #1132.out 11
#1150 errorToCloseZD0208 <= #1132.out 12
#1151 MACRO управление промывкой фильтра ФС02.01.03(pin 1 "сигнал на промывку": #1132.out 1, pin 2 "авария фильтра": DD6_DI.25, pin 3 "подтверждение промывки": DD6_DI.24, pin 4 "сброс аварий": alarmReset, pin 5 "начать очередь снова": filterStartNewQueue, pin 6 "ЗДЭ02.03 открыта": DD7_DI.20, pin 7 "ЗДЭ02.03 закрыта": DD7_DI.21, pin 8 "ЗДЭ02.09 открыта": DD8_DI.0, pin 9 "ЗДЭ02.09 закрыта": DD8_DI.1, pin 10 "время движения ЗДЭ": timeToOpenCloseValve, pin 11 "авария питания ЗДЭ02.03": DD9_DI.6, pin 12 "авария питания ЗДЭ02.09": DD9_DI.12)
	(* <- выход использовать в / последнем фильтре для / начала очереди заново *)
	(* если открыт = промывка *)
	(* если открыт = фильтрация *)
	out 1 "следующий в очереди" <= #1154.output
	out 2 "промыть ФС02.01.03" <= #1153
	#1152 ZD0203:SimpleValve(inputOpen: NOT #1153, inputClose: #1153, statusOpen: pin 6, statusClose: pin 7, reset: pin 4, timeToOpenClose: pin 10)
	out 5 "открыть ЗДЭ02.03" <= #1152.outputOpen
	out 6 "закрыть ЗДЭ02.03" <= #1152.outputClose
	out 7 "авария открытия ЗДЭ02.03" <= #1152.errorToOpen
	#1153 OR(panTestValvesFS020103, #1154.regenFilterOUT)
	out 8 "авария закрытия ЗДЭ02.03" <= #1152.errorToClose
	#1154 FS020103manager:FilterQueueManager(input: pin 1, filterAlarm: #1155, regenFilterStatus: pin 3, alarmReset: pin 4, startNextLoop: pin 5)
	#1155 OR(alarmZD020309, pin 2, pin 11, pin 12)
	#1156 OR(#1152.errorToOpen, #1152.errorToClose, #1158.errorToOpen, #1158.errorToClose)
	#1157 alarmZD020309 <= #1156
	out 3 "ФС02.01.03 промыт" <= #1154.regenerated
	out 4 "не удалось промыть" <= #1154.failToRegen
	#1158 ZD0209:SimpleValve(inputOpen: #1153, inputClose: NOT #1153, statusOpen: pin 8, statusClose: pin 9, reset: pin 4, timeToOpenClose: pin 10)
	out 9 "открыть ЗДЭ02.09" <= #1158.outputOpen
	out 10 "закрыть ЗДЭ02.09" <= #1158.outputClose
	out 11 "авария открытия ЗДЭ02.09" <= #1158.errorToOpen
	out 12 "авария закрытия ЗДЭ02.09" <= #1158.errorToClose
END_MACRO
#1159 DD2_DO.6 <= #1151.out 2
#1160 regeneratedFS020103 <= #1151.out 3
#1161 filterFailToRegen020103 <= #1151.out 4
#1162 DD2_DO.20 <= #1151.out 5
#1163 DD2_DO.21 <= #1151.out 6
#1164 errorToOpenZD0203 <= #1151.out 7
#1165 errorToCloseZD0203 <= #1151.out 8
#1166 DD3_DO.0 <= #1151.out 9
#1167 DD3_DO.1 <= #1151.out 10
#1168 errorToOpenZD0209 <= #1151.out 11
#1169 errorToCloseZD0209 <= #1151.out 12
#1170 MACRO управление промывкой фильтра ФС02.01.04(pin 1 "сигнал на промывку": #1151.out 1, pin 2 "авария фильтра": DD6_DI.27, pin 3 "подтверждение промывки": DD6_DI.26, pin 4 "сброс аварий": alarmReset, pin 5 "начать очередь снова": filterStartNewQueue, pin 6 "ЗДЭ02.04 открыта": DD7_DI.22, pin 7 "ЗДЭ02.04 закрыта": DD7_DI.23, pin 8 "ЗДЭ02.10 открыта": DD8_DI.2, pin 9 "ЗДЭ02.10 закрыта": DD8_DI.3, pin 10 "время движения ЗДЭ": timeToOpenCloseValve, pin 11 "авария питания ЗДЭ02.04": DD9_DI.7, pin 12 "авария питания ЗДЭ02.10": DD9_DI.13)
	(* <- выход использовать в / последнем фильтре для / начала очереди заново *)
	(* если открыт = промывка *)
	(* если открыт = фильтрация *)
	out 1 "следующий в очереди" <= #1173.output
	out 2 "промыть ФС02.01.04" <= #1172
	#1171 ZD0204:SimpleValve(inputOpen: NOT #1172, inputClose: #1172, statusOpen: pin 6, statusClose: pin 7, reset: pin 4, timeToOpenClose: pin 10)
	out 5 "открыть ЗДЭ02.04" <= #1171.outputOpen
	out 6 "закрыть ЗДЭ02.04" <= #1171.outputClose
	out 7 "авария открытия ЗДЭ02.04" <= #1171.errorToOpen
	#1172 OR(panTestValvesFS020104, #1173.regenFilterOUT)
	out 8 "авария закрытия ЗДЭ02.04" <= #1171.errorToClose
	#1173 FS020104manager:FilterQueueManager(input: pin 1, filterAlarm: #1174, regenFilterStatus: pin 3, alarmReset: pin 4, startNextLoop: pin 5)
	#1174 OR(alarmZD020410, pin 2, pin 11, pin 12)
	#1175 OR(#1171.errorToOpen, #1171.errorToClose, #1177.errorToOpen, #1177.errorToClose)
	#1176 alarmZD020410 <= #1175
	out 3 "ФС02.01.04 промыт" <= #1173.regenerated
	out 4 "не удалось промыть" <= #1173.failToRegen
	#1177 ZD0210:SimpleValve(inputOpen: #1172, inputClose: NOT #1172, statusOpen: pin 8, statusClose: pin 9, reset: pin 4, timeToOpenClose: pin 10)
	out 9 "открыть ЗДЭ02.10" <= #1177.outputOpen
	out 10 "закрыть ЗДЭ02.10" <= #1177.outputClose
	out 11 "авария открытия ЗДЭ02.10" <= #1177.errorToOpen
	out 12 "авария закрытия ЗДЭ02.10" <= #1177.errorToClose
END_MACRO
#1178 DD2_DO.7 <= #1170.out 2
#1179 regeneratedFS020104 <= #1170.out 3
#1180 filterFailToRegen020104 <= #1170.out 4
#1181 DD2_DO.22 <= #1170.out 5
#1182 DD2_DO.23 <= #1170.out 6
#1183 errorToOpenZD0204 <= #1170.out 7
#1184 errorToCloseZD0204 <= #1170.out 8
#1185 DD3_DO.2 <= #1170.out 9
#1186 DD3_DO.3 <= #1170.out 10
#1187 errorToOpenZD0210 <= #1170.out 11
#1188 errorToCloseZD0210 <= #1170.out 12
#1189 MACRO управление промывкой фильтра ФС02.01.05(pin 1 "сигнал на промывку": #1170.out 1, pin 2 "авария фильтра": DD6_DI.29, pin 3 "подтверждение промывки": DD6_DI.28, pin 4 "сброс аварий": alarmReset, pin 5 "начать очередь снова": filterStartNewQueue, pin 6 "ЗДЭ02.05 открыта": DD7_DI.24, pin 7 "ЗДЭ02.05 закрыта": DD7_DI.25, pin 8 "ЗДЭ02.11 открыта": DD8_DI.4, pin 9 "ЗДЭ02.11 закрыта": DD8_DI.5, pin 10 "время движения ЗДЭ": timeToOpenCloseValve, pin 11 "авария питания ЗДЭ02.05": DD9_DI.8, pin 12 "авария питания ЗДЭ02.11": DD9_DI.14)
	(* <- выход использовать в / последнем фильтре для / начала очереди заново *)
	(* если открыт = промывка *)
	(* если открыт = фильтрация *)
	out 1 "следующий в очереди" <= #1192.output
	out 2 "промыть ФС02.01.05" <= #1191
	#1190 ZD0205:SimpleValve(inputOpen: NOT #1191, inputClose: #1191, statusOpen: pin 6, statusClose: pin 7, reset: pin 4, timeToOpenClose: pin 10)
	out 5 "открыть ЗДЭ02.05" <= #1190.outputOpen
	out 6 "закрыть ЗДЭ02.05" <= #1190.outputClose
	out 7 "авария открытия ЗДЭ02.05" <= #1190.errorToOpen
	#1191 OR(panTestValvesFS020105, #1192.regenFilterOUT)
	out 8 "авария закрытия ЗДЭ02.05" <= #1190.errorToClose
	#1192 FS020105manager:FilterQueueManager(input: pin 1, filterAlarm: #1193, regenFilterStatus: pin 3, alarmReset: pin 4, startNextLoop: pin 5)
	#1193 OR(alarmZD020511, pin 2, pin 11, pin 12)
	#1194 OR(#1190.errorToOpen, #1190.errorToClose, #1196.errorToOpen, #1196.errorToClose)
	#1195 alarmZD020511 <= #1194
	out 3 "ФС02.01.05 промыт" <= #1192.regenerated
	out 4 "не удалось промыть" <= #1192.failToRegen
	#1196 ZD0211:SimpleValve(inputOpen: #1191, inputClose: NOT #1191, statusOpen: pin 8, statusClose: pin 9, reset: pin 4, timeToOpenClose: pin 10)
	out 9 "открыть ЗДЭ02.11" <= #1196.outputOpen
	out 10 "закрыть ЗДЭ02.11" <= #1196.outputClose
	out 11 "авария открытия ЗДЭ02.11" <= #1196.errorToOpen
	out 12 "авария закрытия ЗДЭ02.11" <= #1196.errorToClose
END_MACRO
#1197 DD2_DO.8 <= #1189.out 2
#1198 regeneratedFS020105 <= #1189.out 3
#1199 filterFailToRegen020105 <= #1189.out 4
#1200 DD2_DO.24 <= #1189.out 5
#1201 DD2_DO.25 <= #1189.out 6
#1202 errorToOpenZD0205 <= #1189.out 7
#1203 errorToCloseZD0205 <= #1189.out 8
#1204 DD3_DO.4 <= #1189.out 9
#1205 DD3_DO.5 <= #1189.out 10
#1206 errorToOpenZD0211 <= #1189.out 11
#1207 errorToCloseZD0211 <= #1189.out 12
#1208 MACRO управление промывкой фильтра ФС02.01.06(pin 1 "сигнал на промывку": #1189.out 1, pin 2 "авария фильтра": DD6_DI.31, pin 3 "подтверждение промывки": DD6_DI.30, pin 4 "сброс аварий": alarmReset, pin 5 "начать очередь снова": filterStartNewQueue, pin 6 "ЗДЭ02.06 открыта": DD7_DI.26, pin 7 "ЗДЭ02.06 закрыта": DD7_DI.27, pin 8 "ЗДЭ02.12 открыта": DD8_DI.6, pin 9 "ЗДЭ02.12 закрыта": DD8_DI.7, pin 10 "время движения ЗДЭ": timeToOpenCloseValve, pin 11 "авария питания ЗДЭ02.06": DD9_DI.9, pin 12 "авария питания ЗДЭ02.12": DD9_DI.15)
	(* <- выход использовать в / последнем фильтре для / начала очереди заново *)
	(* если открыт = промывка *)
	(* если открыт = фильтрация *)
	out 1 "следующий в очереди" <= #1211.output
	out 2 "промыть ФС02.01.06" <= #1210
	#1209 ZD0206:SimpleValve(inputOpen: NOT #1210, inputClose: #1210, statusOpen: pin 6, statusClose: pin 7, reset: pin 4, timeToOpenClose: pin 10)
	out 5 "открыть ЗДЭ02.06" <= #1209.outputOpen
	out 6 "закрыть ЗДЭ02.06" <= #1209.outputClose
	out 7 "авария открытия ЗДЭ02.06" <= #1209.errorToOpen
	#1210 OR(panTestValvesFS020106, #1211.regenFilterOUT)
	out 8 "авария закрытия ЗДЭ02.06" <= #1209.errorToClose
	#1211 FS020106manager:FilterQueueManager(input: pin 1, filterAlarm: #1212, regenFilterStatus: pin 3, alarmReset: pin 4, startNextLoop: pin 5)
	#1212 OR(alarmZD020612, pin 2, pin 11, pin 12)
	#1213 OR(#1209.errorToOpen, #1209.errorToClose, #1215.errorToOpen, #1215.errorToClose)
	#1214 alarmZD020612 <= #1213
	out 3 "ФС02.01.06 промыт" <= #1211.regenerated
	out 4 "не удалось промыть" <= #1211.failToRegen
	#1215 ZD0212:SimpleValve(inputOpen: #1210, inputClose: NOT #1210, statusOpen: pin 8, statusClose: pin 9, reset: pin 4, timeToOpenClose: pin 10)
	out 9 "открыть ЗДЭ02.12" <= #1215.outputOpen
	out 10 "закрыть ЗДЭ02.12" <= #1215.outputClose
	out 11 "авария открытия ЗДЭ02.12" <= #1215.errorToOpen
	out 12 "авария закрытия ЗДЭ02.12" <= #1215.errorToClose
END_MACRO
#1216 DD2_DO.9 <= #1208.out 2
#1217 regeneratedFS020106 <= #1208.out 3
#1218 filterFailToRegen020106 <= #1208.out 4
#1219 DD2_DO.26 <= #1208.out 5
#1220 DD2_DO.27 <= #1208.out 6
#1221 errorToOpenZD0206 <= #1208.out 7
#1222 errorToCloseZD0206 <= #1208.out 8
#1223 DD3_DO.6 <= #1208.out 9
#1224 DD3_DO.7 <= #1208.out 10
#1225 errorToOpenZD0212 <= #1208.out 11
#1226 errorToCloseZD0212 <= #1208.out 12
#1227 MACRO управление промывкой фильтра ФС02.02.01(pin 1 "сигнал на промывку": #1208.out 1, pin 2 "авария фильтра": DD7_DI.1, pin 3 "подтверждение промывки": DD7_DI.0, pin 4 "сброс аварий": alarmReset, pin 5 "начать очередь снова": filterStartNewQueue, pin 6 "ЗДЭ02.13 открыта": DD8_DI.8, pin 7 "ЗДЭ02.13 закрыта": DD8_DI.9, pin 8 "ЗДЭ02.19 открыта": DD8_DI.20, pin 9 "ЗДЭ02.19 закрыта": DD8_DI.21, pin 10 "время движения ЗДЭ": timeToOpenCloseValve, pin 11 "авария питания ЗДЭ02.13": DD9_DI.16, pin 12 "авария питания ЗДЭ02.19": DD9_DI.22)
	(* <- выход использовать в / последнем фильтре для / начала очереди заново *)
	(* если открыт = промывка *)
	(* если открыт = фильтрация *)
	out 1 "следующий в очереди" <= #1230.output
	out 2 "промыть ФС02.02.01" <= #1229
	#1228 ZD0213:SimpleValve(inputOpen: NOT #1229, inputClose: #1229, statusOpen: pin 6, statusClose: pin 7, reset: pin 4, timeToOpenClose: pin 10)
